C07299=1201.036,66.508,-47.398,-179.072,5.766,148.745
C07300=1201.040,66.258,-47.381,-179.075,5.765,148.746
C07301=1201.046,66.009,-47.364,-179.078,5.764,148.746
C07302=1201.050,65.759,-47.347,-179.080,5.763,148.747
C07303=1201.056,65.510,-47.330,-179.083,5.762,148.747
C07304=1201.060,65.261,-47.313,-179.086,5.762,148.748
C07305=1201.065,65.012,-47.296,-179.088,5.761,148.748
C07306=1201.070,64.763,-47.279,-179.090,5.760,148.749
C07307=1201.075,64.513,-47.263,-179.093,5.760,148.750
C07308=1201.080,64.263,-47.245,-179.096,5.758,148.750
C07309=1201.085,64.014,-47.229,-179.098,5.757,148.751
C07310=1201.090,63.765,-47.212,-179.101,5.757,148.751
C07311=1201.095,63.515,-47.195,-179.103,5.756,148.752
C07312=1201.099,63.266,-47.178,-179.106,5.755,148.753
C07313=1201.104,63.017,-47.162,-179.109,5.754,148.753
C07314=1201.110,62.767,-47.145,-179.111,5.753,148.754
C07315=1201.114,62.518,-47.128,-179.114,5.753,148.754
C07316=1201.119,62.268,-47.111,-179.116,5.752,148.755
C07317=1201.124,62.019,-47.095,-179.119,5.751,148.756
C07318=1201.129,61.770,-47.078,-179.121,5.751,148.756
C07319=1201.134,61.519,-47.062,-179.124,5.749,148.757
C07320=1201.140,61.270,-47.045,-179.127,5.749,148.757
C07321=1201.144,61.021,-47.028,-179.129,5.748,148.758
C07322=1201.149,60.771,-47.012,-179.132,5.747,148.758
C07323=1201.154,60.522,-46.995,-179.134,5.747,148.759
C07324=1201.159,60.273,-46.978,-179.137,5.746,148.760
C07325=1201.164,60.024,-46.962,-179.140,5.744,148.760
C07326=1201.168,59.775,-46.945,-179.142,5.744,148.761
C07327=1201.174,59.525,-46.928,-179.145,5.743,148.761
C07328=1201.179,59.276,-46.912,-179.147,5.742,148.762
C07329=1201.183,59.026,-46.896,-179.150,5.742,148.763
C07330=1201.188,58.776,-46.879,-179.152,5.741,148.763
C07331=1201.194,58.527,-46.862,-179.155,5.740,148.764
C07332=1201.198,58.278,-46.845,-179.158,5.739,148.764
C07333=1201.203,58.029,-46.829,-179.160,5.738,148.765
C07334=1201.208,57.779,-46.813,-179.163,5.738,148.766
C07335=1201.213,57.529,-46.796,-179.165,5.737,148.766
C07336=1201.218,57.280,-46.780,-179.168,5.736,148.767
C07337=1201.223,57.031,-46.763,-179.170,5.736,148.767
C07338=1201.228,56.782,-46.747,-179.173,5.734,148.768
C07339=1201.233,56.532,-46.731,-179.176,5.734,148.769
C07340=1201.238,56.282,-46.713,-179.178,5.733,148.769
C07341=1201.243,56.033,-46.697,-179.181,5.732,148.770
C07342=1201.248,55.784,-46.680,-179.183,5.732,148.770
C07343=1201.253,55.534,-46.665,-179.186,5.731,148.771
C07344=1201.258,55.266,-46.647,-179.189,5.729,148.772
C07345=1201.264,54.997,-46.629,-179.191,5.729,148.772
C07346=1201.269,54.729,-46.611,-179.194,5.728,148.773
C07347=1201.274,54.460,-46.594,-179.197,5.727,148.774
C07348=1201.279,54.211,-46.578,-179.200,5.726,148.774
C07349=1201.284,53.962,-46.561,-179.202,5.726,148.775
C07350=1201.288,53.712,-46.545,-179.204,5.725,148.775
C07351=1201.294,53.463,-46.528,-179.207,5.724,148.776
C07352=1201.299,53.213,-46.512,-179.210,5.724,148.777
C07353=1201.304,52.964,-46.496,-179.212,5.723,148.777
C07354=1201.309,52.714,-46.479,-179.215,5.722,148.778
C07355=1201.314,52.465,-46.464,-179.218,5.721,148.778
C07356=1201.318,52.215,-46.447,-179.220,5.721,148.779
C07357=1201.324,51.967,-46.431,-179.223,5.720,148.780
C07358=1201.328,51.716,-46.415,-179.225,5.719,148.780
C07359=1201.333,51.468,-46.398,-179.228,5.719,148.781
C07360=1201.338,51.218,-46.383,-179.230,5.718,148.781
C07361=1201.343,50.969,-46.366,-179.233,5.717,148.782
C07362=1201.348,50.719,-46.350,-179.235,5.717,148.783
C07363=1201.353,50.470,-46.334,-179.238,5.716,148.783
C07364=1201.358,50.220,-46.317,-179.241,5.714,148.784
C07365=1201.364,49.971,-46.301,-179.243,5.714,148.784
C07366=1201.368,49.721,-46.284,-179.246,5.713,148.785
C07367=1201.374,49.472,-46.269,-179.249,5.713,148.786
C07368=1201.378,49.222,-46.252,-179.251,5.712,148.786
C07369=1201.383,48.973,-46.237,-179.253,5.711,148.787
C07370=1201.388,48.723,-46.220,-179.256,5.711,148.788
C07371=1201.393,48.474,-46.204,-179.258,5.710,148.788
C07372=1201.398,48.225,-46.188,-179.261,5.709,148.789
C07373=1201.403,47.975,-46.172,-179.264,5.708,148.789
C07374=1201.408,47.725,-46.156,-179.267,5.708,148.790
C07375=1201.412,47.477,-46.140,-179.269,5.707,148.790
C07376=1201.418,47.227,-46.125,-179.271,5.706,148.791
C07377=1201.422,46.978,-46.108,-179.274,5.706,148.792
C07378=1201.428,46.728,-46.093,-179.277,5.705,148.792
C07379=1201.432,46.479,-46.076,-179.279,5.704,148.793
C07380=1201.437,46.229,-46.060,-179.281,5.704,148.794
C07381=1201.442,45.979,-46.044,-179.284,5.703,148.794
C07382=1201.447,45.731,-46.028,-179.286,5.702,148.795
C07383=1201.453,45.481,-46.012,-179.289,5.702,148.795
C07384=1201.458,45.231,-45.997,-179.292,5.700,148.796
C07385=1201.463,44.982,-45.980,-179.295,5.700,148.797
C07386=1201.467,44.732,-45.964,-179.297,5.699,148.797
C07387=1201.472,44.483,-45.948,-179.300,5.698,148.798
C07388=1201.478,44.234,-45.932,-179.302,5.698,148.798
C07389=1201.482,43.984,-45.917,-179.305,5.697,148.799
C07390=1201.487,43.735,-45.901,-179.307,5.696,148.800
C07391=1201.492,43.485,-45.885,-179.310,5.696,148.800
C07392=1201.497,43.236,-45.869,-179.312,5.695,148.801
C07393=1201.503,42.986,-45.854,-179.315,5.695,148.802
C07394=1201.507,42.737,-45.837,-179.317,5.694,148.802
C07395=1201.512,42.488,-45.821,-179.320,5.693,148.803
C07396=1201.518,42.238,-45.806,-179.322,5.693,148.803
C07397=1201.522,41.988,-45.790,-179.325,5.692,148.804
C07398=1201.527,41.740,-45.774,-179.328,5.691,148.804
C07399=1201.532,41.490,-45.758,-179.330,5.690,148.805
C07400=1201.537,41.240,-45.743,-179.333,5.690,148.806
C07401=1201.542,40.991,-45.727,-179.336,5.689,148.806
C07402=1201.547,40.741,-45.710,-179.338,5.688,148.807
C07403=1201.552,40.492,-45.695,-179.340,5.688,148.808
C07404=1201.557,40.243,-45.680,-179.343,5.687,148.808
C07405=1201.562,39.993,-45.664,-179.346,5.687,148.809
C07406=1201.567,39.743,-45.648,-179.348,5.686,148.809
C07407=1201.572,39.494,-45.633,-179.350,5.685,148.810
C07408=1201.577,39.245,-45.617,-179.353,5.685,148.811
C07409=1201.582,38.995,-45.601,-179.356,5.684,148.811
C07410=1201.587,38.746,-45.585,-179.358,5.683,148.812
C07411=1201.592,38.496,-45.570,-179.361,5.683,148.813
C07412=1201.597,38.247,-45.554,-179.363,5.682,148.813
C07413=1201.602,37.997,-45.539,-179.366,5.682,148.814
C07414=1201.607,37.748,-45.523,-179.368,5.681,148.814
C07415=1201.612,37.498,-45.507,-179.371,5.680,148.815
C07416=1201.617,37.249,-45.492,-179.374,5.679,148.816
C07417=1201.622,37.000,-45.476,-179.376,5.678,148.816
C07418=1201.627,36.750,-45.460,-179.379,5.678,148.817
C07419=1201.631,36.501,-45.445,-179.381,5.677,148.817
C07420=1201.637,36.251,-45.429,-179.384,5.676,148.818
C07421=1201.642,36.002,-45.414,-179.387,5.676,148.819
C07422=1201.647,35.752,-45.398,-179.389,5.675,148.820
C07423=1201.651,35.503,-45.383,-179.391,5.674,148.820
C07424=1201.657,35.253,-45.367,-179.394,5.674,148.821
C07425=1201.662,35.004,-45.352,-179.397,5.673,148.821
C07426=1201.667,34.755,-45.337,-179.399,5.673,148.822
C07427=1201.672,34.505,-45.321,-179.401,5.672,148.822
C07428=1201.677,34.255,-45.305,-179.404,5.671,148.823
C07429=1201.682,34.006,-45.290,-179.407,5.671,148.824
C07430=1201.687,33.757,-45.275,-179.409,5.670,148.824
C07431=1201.691,33.507,-45.259,-179.412,5.670,148.825
C07432=1201.697,33.258,-45.244,-179.414,5.669,148.826
C07433=1201.702,33.008,-45.228,-179.417,5.668,148.826
C07434=1201.707,32.759,-45.213,-179.419,5.668,148.827
C07435=1201.712,32.510,-45.197,-179.422,5.667,148.828
C07436=1201.717,32.259,-45.182,-179.424,5.667,148.828
C07437=1201.722,32.010,-45.167,-179.427,5.666,148.829
C07438=1201.727,31.760,-45.152,-179.430,5.665,148.829
C07439=1201.732,31.511,-45.137,-179.432,5.665,148.830
C07440=1201.737,31.262,-45.121,-179.434,5.664,148.831
C07441=1201.742,31.012,-45.105,-179.437,5.664,148.831
C07442=1201.747,30.763,-45.090,-179.440,5.663,148.832
C07443=1201.752,30.513,-45.075,-179.442,5.663,148.833
C07444=1201.757,30.264,-45.060,-179.445,5.662,148.833
C07445=1201.762,30.014,-45.045,-179.447,5.661,148.834
C07446=1201.766,29.764,-45.029,-179.450,5.661,148.834
C07447=1201.772,29.515,-45.014,-179.452,5.660,148.835
C07448=1201.777,29.246,-44.998,-179.455,5.660,148.836
C07449=1201.782,28.978,-44.981,-179.458,5.658,148.836
C07450=1201.788,28.709,-44.965,-179.461,5.658,148.837
C07451=1201.793,28.441,-44.948,-179.464,5.657,148.838
C07452=1201.798,28.191,-44.933,-179.466,5.657,148.838
C07453=1201.803,27.941,-44.918,-179.469,5.656,148.839
C07454=1201.809,27.692,-44.903,-179.471,5.655,148.840
C07455=1201.813,27.443,-44.888,-179.474,5.655,148.840
C07456=1201.818,27.193,-44.872,-179.476,5.654,148.841
C07457=1201.823,26.943,-44.858,-179.479,5.654,148.842
C07458=1201.829,26.694,-44.842,-179.481,5.653,148.842
C07459=1201.833,26.445,-44.827,-179.484,5.652,148.843
C07460=1201.839,26.195,-44.812,-179.486,5.652,148.843
C07461=1201.844,25.946,-44.797,-179.489,5.651,148.844
C07462=1201.849,25.696,-44.782,-179.492,5.651,148.845
C07463=1201.854,25.447,-44.767,-179.494,5.650,148.845
C07464=1201.859,25.197,-44.752,-179.496,5.649,148.846
C07465=1201.863,24.947,-44.736,-179.499,5.649,148.847
C07466=1201.868,24.698,-44.721,-179.502,5.648,148.847
C07467=1201.874,24.448,-44.706,-179.504,5.648,148.848
C07468=1201.878,24.199,-44.691,-179.507,5.647,148.848
C07469=1201.884,23.950,-44.676,-179.509,5.646,148.849
C07470=1201.889,23.700,-44.662,-179.512,5.646,148.850
C07471=1201.893,23.451,-44.647,-179.514,5.645,148.850
C07472=1201.899,23.201,-44.632,-179.517,5.645,148.851
C07473=1201.904,22.952,-44.617,-179.519,5.645,148.852
C07474=1201.908,22.703,-44.602,-179.521,5.644,148.852
C07475=1201.914,22.453,-44.587,-179.524,5.644,148.853
C07476=1201.919,22.203,-44.572,-179.527,5.643,148.854
C07477=1201.924,21.953,-44.557,-179.529,5.643,148.854
C07478=1201.929,21.704,-44.542,-179.531,5.642,148.855
C07479=1201.933,21.454,-44.527,-179.534,5.641,148.855
C07480=1201.939,21.205,-44.512,-179.537,5.641,148.856
C07481=1201.943,20.955,-44.497,-179.539,5.640,148.857
C07482=1201.948,20.706,-44.483,-179.542,5.640,148.857
C07483=1201.954,20.456,-44.467,-179.544,5.639,148.858
C07484=1201.959,20.207,-44.453,-179.547,5.638,148.859
C07485=1201.963,19.958,-44.438,-179.549,5.638,148.859
C07486=1201.969,19.708,-44.423,-179.552,5.637,148.860
C07487=1201.974,19.458,-44.408,-179.555,5.637,148.861
C07488=1201.979,19.209,-44.394,-179.557,5.636,148.861
C07489=1201.984,18.959,-44.378,-179.560,5.636,148.862
C07490=1201.989,18.710,-44.364,-179.562,5.635,148.862
C07491=1201.994,18.460,-44.349,-179.565,5.634,148.863
C07492=1201.999,18.211,-44.334,-179.568,5.634,148.864
C07493=1202.004,17.961,-44.320,-179.570,5.633,148.864
C07494=1202.009,17.712,-44.305,-179.572,5.633,148.865
C07495=1202.014,17.462,-44.290,-179.575,5.632,148.866
C07496=1202.019,17.213,-44.275,-179.577,5.632,148.866
C07497=1202.024,16.963,-44.260,-179.580,5.632,148.867
C07498=1202.029,16.713,-44.246,-179.582,5.631,148.868
C07499=1202.034,16.464,-44.231,-179.585,5.630,148.868
C07500=1202.039,16.215,-44.217,-179.587,5.630,148.869
C07501=1202.045,15.966,-44.202,-179.590,5.629,148.869
C07502=1202.050,15.716,-44.187,-179.592,5.629,148.870
C07503=1202.055,15.466,-44.173,-179.595,5.628,148.871
C07504=1202.059,15.217,-44.158,-179.597,5.628,148.871
C07505=1202.064,14.967,-44.144,-179.600,5.627,148.872
C07506=1202.070,14.717,-44.129,-179.603,5.627,148.873
C07507=1202.075,14.468,-44.114,-179.605,5.626,148.873
C07508=1202.080,14.219,-44.100,-179.608,5.626,148.874
C07509=1202.085,13.969,-44.085,-179.611,5.625,148.875
C07510=1202.089,13.720,-44.070,-179.613,5.624,148.875
C07511=1202.095,13.470,-44.056,-179.615,5.624,148.876
C07512=1202.100,13.220,-44.041,-179.617,5.624,148.877
C07513=1202.105,12.970,-44.027,-179.620,5.623,148.877
C07514=1202.109,12.721,-44.012,-179.623,5.623,148.878
C07515=1202.115,12.472,-43.998,-179.625,5.622,148.878
C07516=1202.120,12.223,-43.984,-179.627,5.622,148.879
C07517=1202.125,11.973,-43.969,-179.630,5.621,148.880
C07518=1202.130,11.723,-43.954,-179.633,5.621,148.880
C07519=1202.135,11.474,-43.940,-179.635,5.620,148.881
C07520=1202.140,11.224,-43.925,-179.638,5.620,148.882
C07521=1202.145,10.974,-43.911,-179.640,5.619,148.882
C07522=1202.150,10.725,-43.896,-179.643,5.618,148.883
C07523=1202.155,10.476,-43.882,-179.646,5.618,148.884
C07524=1202.160,10.227,-43.868,-179.648,5.618,148.884
C07525=1202.165,9.977,-43.854,-179.650,5.617,148.885
C07526=1202.170,9.727,-43.839,-179.652,5.617,148.885
C07527=1202.175,9.477,-43.825,-179.655,5.616,148.886
C07528=1202.181,9.228,-43.809,-179.658,5.616,148.887
C07529=1202.185,8.978,-43.795,-179.660,5.615,148.888
C07530=1202.190,8.729,-43.781,-179.663,5.615,148.888
C07531=1202.196,8.480,-43.767,-179.666,5.614,148.889
C07532=1202.201,8.230,-43.753,-179.668,5.613,148.889
C07533=1202.206,7.980,-43.738,-179.671,5.613,148.890
C07534=1202.211,7.730,-43.724,-179.673,5.613,148.891
C07535=1202.216,7.481,-43.710,-179.675,5.613,148.891
C07536=1202.220,7.232,-43.695,-179.678,5.612,148.892
C07537=1202.226,6.983,-43.681,-179.681,5.612,148.893
C07538=1202.231,6.733,-43.667,-179.683,5.611,148.893
C07539=1202.236,6.483,-43.652,-179.685,5.610,148.894
C07540=1202.241,6.233,-43.638,-179.688,5.610,148.895
C07541=1202.246,5.984,-43.624,-179.691,5.609,148.895
C07542=1202.251,5.735,-43.610,-179.693,5.609,148.896
C07543=1202.256,5.485,-43.596,-179.696,5.608,148.897
C07544=1202.261,5.235,-43.581,-179.698,5.608,148.897
C07545=1202.266,4.986,-43.567,-179.700,5.608,148.898
C07546=1202.271,4.736,-43.553,-179.703,5.607,148.898
C07547=1202.277,4.487,-43.539,-179.705,5.607,148.899
C07548=1202.282,4.237,-43.525,-179.708,5.606,148.900
C07549=1202.287,3.987,-43.510,-179.711,5.606,148.901
C07550=1202.292,3.738,-43.496,-179.713,5.605,148.901
C07551=1202.297,3.489,-43.482,-179.716,5.604,148.902
C07552=1202.303,3.219,-43.467,-179.718,5.604,148.902
C07553=1202.308,2.951,-43.452,-179.721,5.603,148.903
C07554=1202.313,2.681,-43.437,-179.724,5.603,148.904
C07555=1202.319,2.412,-43.422,-179.726,5.602,148.904
C07556=1202.324,2.162,-43.407,-179.729,5.602,148.905
C07557=1202.328,1.913,-43.394,-179.731,5.602,148.906
C07558=1202.333,1.664,-43.380,-179.734,5.602,148.907
C07559=1202.338,1.414,-43.365,-179.736,5.601,148.907
C07560=1202.344,1.165,-43.351,-179.739,5.601,148.908
C07561=1202.349,0.915,-43.337,-179.741,5.600,148.908
C07562=1202.354,0.665,-43.323,-179.744,5.599,148.909
C07563=1202.359,0.415,-43.309,-179.746,5.599,148.910
C07564=1202.365,0.166,-43.295,-179.749,5.598,148.910
C07565=1202.370,-0.084,-43.281,-179.751,5.599,148.911
C07566=1202.374,-0.333,-43.267,-179.754,5.598,148.912
C07567=1202.379,-0.582,-43.254,-179.756,5.598,148.912
C07568=1202.384,-0.832,-43.239,-179.759,5.597,148.913
C07569=1202.389,-1.081,-43.225,-179.761,5.596,148.914
C07570=1202.394,-1.332,-43.211,-179.764,5.596,148.914
C07571=1202.400,-1.581,-43.198,-179.767,5.595,148.915
C07572=1202.404,-1.830,-43.184,-179.769,5.596,148.916
C07573=1202.409,-2.080,-43.170,-179.771,5.595,148.916
C07574=1202.415,-2.329,-43.156,-179.773,5.594,148.917
C07575=1202.420,-2.579,-43.142,-179.776,5.594,148.918
C07576=1202.425,-2.829,-43.128,-179.779,5.593,148.918
C07577=1202.430,-3.078,-43.115,-179.781,5.593,148.919
C07578=1202.435,-3.327,-43.100,-179.784,5.592,148.920
C07579=1202.440,-3.578,-43.087,-179.786,5.593,148.920
C07580=1202.446,-3.827,-43.073,-179.788,5.592,148.921
C07581=1202.450,-4.076,-43.059,-179.791,5.591,148.921
C07582=1202.455,-4.326,-43.046,-179.794,5.591,148.922
C07583=1202.461,-4.575,-43.032,-179.796,5.590,148.923
C07584=1202.466,-4.825,-43.017,-179.799,5.590,148.924
C07585=1202.470,-5.075,-43.004,-179.801,5.590,148.924
C07586=1202.476,-5.324,-42.990,-179.804,5.590,148.925
C07587=1202.481,-5.574,-42.976,-179.806,5.589,148.925
C07588=1202.486,-5.823,-42.962,-179.808,5.588,148.926
C07589=1202.491,-6.073,-42.949,-179.811,5.588,148.927
C07590=1202.496,-6.323,-42.935,-179.814,5.587,148.927
C07591=1202.501,-6.572,-42.921,-179.816,5.588,148.928
C07592=1202.506,-6.822,-42.908,-179.819,5.587,148.929
C07593=1202.511,-7.071,-42.894,-179.821,5.586,148.929
C07594=1202.517,-7.321,-42.881,-179.823,5.586,148.930
C07595=1202.521,-7.571,-42.866,-179.826,5.585,148.931
C07596=1202.526,-7.819,-42.853,-179.829,5.585,148.931
C07597=1202.532,-8.070,-42.840,-179.831,5.585,148.932
C07598=1202.537,-8.319,-42.825,-179.833,5.585,148.933
C07599=1202.542,-8.569,-42.813,-179.836,5.584,148.933
C07600=1202.547,-8.818,-42.798,-179.838,5.583,148.934
C07601=1202.552,-9.067,-42.784,-179.841,5.583,148.935
C07602=1202.557,-9.317,-42.771,-179.844,5.582,148.935
C07603=1202.562,-9.566,-42.758,-179.846,5.583,148.936
C07604=1202.567,-9.817,-42.744,-179.848,5.582,148.937
C07605=1202.572,-10.066,-42.730,-179.851,5.582,148.937
C07606=1202.578,-10.316,-42.717,-179.854,5.581,148.938
C07607=1202.582,-10.565,-42.703,-179.856,5.580,148.938
C07608=1202.588,-10.815,-42.690,-179.858,5.580,148.939
C07609=1202.593,-11.065,-42.676,-179.860,5.580,148.940
C07610=1202.598,-11.314,-42.663,-179.863,5.580,148.941
C07611=1202.603,-11.564,-42.649,-179.866,5.579,148.941
C07612=1202.607,-11.814,-42.636,-179.868,5.579,148.942
C07613=1202.613,-12.063,-42.622,-179.871,5.578,148.942
C07614=1202.618,-12.313,-42.609,-179.873,5.578,148.943
C07615=1202.623,-12.562,-42.595,-179.875,5.578,148.944
C07616=1202.628,-12.812,-42.582,-179.878,5.577,148.944
C07617=1202.633,-13.061,-42.568,-179.881,5.577,148.945
C07618=1202.638,-13.311,-42.555,-179.883,5.576,148.946
C07619=1202.643,-13.560,-42.542,-179.885,5.576,148.947
C07620=1202.648,-13.810,-42.528,-179.888,5.576,148.947
C07621=1202.653,-14.059,-42.515,-179.890,5.575,148.948
C07622=1202.658,-14.309,-42.501,-179.893,5.575,148.948
C07623=1202.664,-14.559,-42.488,-179.896,5.574,148.949
C07624=1202.668,-14.808,-42.474,-179.898,5.574,148.950
C07625=1202.674,-15.058,-42.461,-179.900,5.574,148.951
C07626=1202.679,-15.308,-42.448,-179.903,5.574,148.951
C07627=1202.684,-15.557,-42.434,-179.905,5.573,148.952
C07628=1202.689,-15.807,-42.421,-179.908,5.572,148.952
C07629=1202.695,-16.056,-42.408,-179.910,5.572,148.953
C07630=1202.699,-16.306,-42.394,-179.912,5.572,148.954
C07631=1202.705,-16.555,-42.381,-179.915,5.572,148.954
C07632=1202.709,-16.805,-42.368,-179.918,5.571,148.955
C07633=1202.715,-17.054,-42.354,-179.920,5.571,148.956
C07634=1202.720,-17.304,-42.342,-179.922,5.571,148.956
C07635=1202.725,-17.554,-42.328,-179.925,5.570,148.957
C07636=1202.730,-17.803,-42.315,-179.927,5.570,148.958
C07637=1202.735,-18.053,-42.302,-179.930,5.569,148.958
C07638=1202.740,-18.302,-42.289,-179.933,5.569,148.959
C07639=1202.745,-18.552,-42.276,-179.935,5.569,148.960
C07640=1202.751,-18.801,-42.262,-179.937,5.568,148.960
C07641=1202.755,-19.051,-42.249,-179.940,5.568,148.961
C07642=1202.761,-19.301,-42.236,-179.942,5.567,148.962
C07643=1202.766,-19.550,-42.223,-179.944,5.567,148.962
C07644=1202.771,-19.800,-42.209,-179.947,5.567,148.963
C07645=1202.776,-20.049,-42.196,-179.950,5.566,148.964
C07646=1202.781,-20.299,-42.183,-179.952,5.566,148.964
C07647=1202.787,-20.549,-42.170,-179.955,5.566,148.965
C07648=1202.792,-20.798,-42.157,-179.957,5.565,148.966
C07649=1202.797,-21.048,-42.143,-179.959,5.565,148.966
C07650=1202.802,-21.297,-42.130,-179.962,5.565,148.967
C07651=1202.806,-21.547,-42.118,-179.964,5.564,148.968
C07652=1202.812,-21.797,-42.104,-179.967,5.564,148.968
C07653=1202.817,-22.046,-42.092,-179.969,5.564,148.969
C07654=1202.821,-22.296,-42.078,-179.972,5.563,148.970
C07655=1202.827,-22.545,-42.065,-179.974,5.563,148.970
C07656=1202.832,-22.815,-42.051,-179.977,5.562,148.971
C07657=1202.838,-23.085,-42.037,-179.980,5.562,148.972
C07658=1202.844,-23.355,-42.023,-179.982,5.562,148.973
C07659=1202.849,-23.624,-42.009,-179.985,5.562,148.973
C07660=1202.854,-23.873,-41.996,-179.987,5.561,148.974
C07661=1202.859,-24.123,-41.982,-179.989,5.561,148.974
C07662=1202.865,-24.373,-41.970,-179.992,5.560,148.975
C07663=1202.870,-24.622,-41.957,-179.994,5.560,148.976
C07664=1202.875,-24.872,-41.944,-179.997,5.560,148.976
C07665=1202.880,-25.122,-41.931,-180.000,5.559,148.977
C07666=1202.885,-25.371,-41.918,179.998,5.559,148.978
C07667=1202.890,-25.621,-41.905,179.996,5.559,148.979
C07668=1202.896,-25.871,-41.892,179.994,5.558,148.979
C07669=1202.900,-26.121,-41.879,179.991,5.558,148.980
C07670=1202.905,-26.370,-41.867,179.988,5.558,148.980
C07671=1202.911,-26.620,-41.854,179.986,5.558,148.981
C07672=1202.916,-26.869,-41.841,179.984,5.557,148.982
C07673=1202.921,-27.119,-41.828,179.981,5.557,148.983
C07674=1202.926,-27.368,-41.815,179.978,5.556,148.983
C07675=1202.932,-27.618,-41.802,179.976,5.557,148.984
C07676=1202.936,-27.868,-41.789,179.974,5.556,148.984
C07677=1202.941,-28.117,-41.777,179.971,5.555,148.985
C07678=1202.947,-28.366,-41.764,179.969,5.555,148.986
C07679=1202.951,-28.616,-41.751,179.967,5.555,148.986
C07680=1202.957,-28.866,-41.738,179.964,5.555,148.987
C07681=1202.962,-29.115,-41.725,179.961,5.554,148.988
C07682=1202.967,-29.365,-41.712,179.959,5.554,148.989
C07683=1202.972,-29.615,-41.700,179.957,5.554,148.989
C07684=1202.978,-29.864,-41.686,179.954,5.553,148.990
C07685=1202.983,-30.114,-41.674,179.952,5.553,148.990
C07686=1202.987,-30.364,-41.661,179.949,5.552,148.991
C07687=1202.992,-30.613,-41.648,179.947,5.553,148.992
C07688=1202.997,-30.862,-41.636,179.944,5.552,148.993
C07689=1203.003,-31.112,-41.623,179.942,5.552,148.993
C07690=1203.008,-31.363,-41.610,179.939,5.551,148.994
C07691=1203.013,-31.612,-41.598,179.937,5.551,148.994
C07692=1203.018,-31.861,-41.585,179.935,5.551,148.995
C07693=1203.024,-32.111,-41.572,179.932,5.550,148.996
C07694=1203.028,-32.361,-41.559,179.929,5.550,148.996
C07695=1203.033,-32.610,-41.547,179.927,5.550,148.997
C07696=1203.038,-32.859,-41.534,179.925,5.550,148.998
C07697=1203.044,-33.109,-41.522,179.922,5.549,148.998
C07698=1203.049,-33.360,-41.509,179.920,5.549,148.999
C07699=1203.054,-33.609,-41.496,179.918,5.549,149.000
C07700=1203.059,-33.858,-41.484,179.915,5.548,149.000
C07701=1203.064,-34.107,-41.471,179.912,5.548,149.001
C07702=1203.070,-34.357,-41.459,179.910,5.548,149.002
C07703=1203.074,-34.607,-41.446,179.908,5.548,149.003
C07704=1203.079,-34.857,-41.434,179.905,5.547,149.003
C07705=1203.085,-35.106,-41.421,179.903,5.547,149.004
C07706=1203.091,-35.356,-41.409,179.901,5.547,149.004
C07707=1203.096,-35.606,-41.396,179.898,5.546,149.005
C07708=1203.100,-35.856,-41.383,179.895,5.546,149.006
C07709=1203.105,-36.105,-41.370,179.893,5.546,149.006
C07710=1203.111,-36.355,-41.358,179.891,5.546,149.007
C07711=1203.116,-36.604,-41.346,179.888,5.545,149.008
C07712=1203.121,-36.854,-41.333,179.886,5.545,149.008
C07713=1203.126,-37.104,-41.320,179.884,5.545,149.009
C07714=1203.131,-37.353,-41.308,179.881,5.544,149.010
C07715=1203.136,-37.603,-41.296,179.878,5.544,149.010
C07716=1203.141,-37.852,-41.283,179.876,5.544,149.011
C07717=1203.147,-38.102,-41.271,179.874,5.544,149.012
C07718=1203.152,-38.351,-41.259,179.871,5.543,149.012
C07719=1203.157,-38.601,-41.246,179.869,5.543,149.013
C07720=1203.162,-38.851,-41.234,179.867,5.543,149.014
C07721=1203.167,-39.101,-41.221,179.864,5.542,149.014
C07722=1203.172,-39.350,-41.209,179.861,5.542,149.015
C07723=1203.178,-39.600,-41.197,179.859,5.542,149.016
C07724=1203.183,-39.849,-41.184,179.857,5.542,149.017
C07725=1203.188,-40.099,-41.172,179.855,5.541,149.017
C07726=1203.193,-40.348,-41.160,179.852,5.541,149.018
C07727=1203.198,-40.598,-41.147,179.850,5.541,149.018
C07728=1203.203,-40.848,-41.135,179.847,5.540,149.019
C07729=1203.208,-41.098,-41.122,179.845,5.541,149.020
C07730=1203.214,-41.348,-41.110,179.842,5.540,149.021
C07731=1203.219,-41.597,-41.098,179.840,5.540,149.021
C07732=1203.224,-41.846,-41.085,179.838,5.539,149.022
C07733=1203.229,-42.096,-41.073,179.835,5.539,149.022
C07734=1203.235,-42.346,-41.061,179.833,5.539,149.023
C07735=1203.240,-42.595,-41.049,179.830,5.538,149.024
C07736=1203.244,-42.846,-41.036,179.828,5.539,149.024
C07737=1203.249,-43.095,-41.025,179.825,5.538,149.025
C07738=1203.254,-43.344,-41.012,179.823,5.538,149.026
C07739=1203.260,-43.594,-41.000,179.821,5.538,149.026
C07740=1203.265,-43.844,-40.987,179.818,5.537,149.027
C07741=1203.270,-44.094,-40.976,179.816,5.537,149.028
C07742=1203.275,-44.343,-40.963,179.814,5.537,149.028
C07743=1203.281,-44.593,-40.951,179.811,5.537,149.029
C07744=1203.286,-44.842,-40.938,179.808,5.536,149.030
C07745=1203.291,-45.092,-40.927,179.806,5.535,149.030
C07746=1203.296,-45.341,-40.915,179.804,5.536,149.031
C07747=1203.301,-45.591,-40.903,179.801,5.535,149.032
C07748=1203.306,-45.840,-40.890,179.799,5.535,149.032
C07749=1203.312,-46.090,-40.878,179.797,5.535,149.033
C07750=1203.317,-46.340,-40.866,179.794,5.535,149.034
C07751=1203.322,-46.590,-40.854,179.791,5.534,149.035
C07752=1203.327,-46.840,-40.841,179.790,5.534,149.035
C07753=1203.332,-47.089,-40.829,179.787,5.534,149.036
C07754=1203.337,-47.339,-40.818,179.784,5.533,149.036
C07755=1203.342,-47.589,-40.806,179.782,5.534,149.037
C07756=1203.347,-47.838,-40.793,179.780,5.533,149.038
C07757=1203.353,-48.088,-40.781,179.777,5.533,149.039
C07758=1203.357,-48.337,-40.769,179.775,5.533,149.039
C07759=1203.363,-48.587,-40.757,179.773,5.532,149.040
C07760=1203.369,-48.857,-40.745,179.770,5.532,149.040
C07761=1203.375,-49.128,-40.731,179.767,5.532,149.041
C07762=1203.380,-49.398,-40.718,179.765,5.532,149.042
C07763=1203.386,-49.668,-40.706,179.762,5.532,149.043
C07764=1203.391,-49.917,-40.693,179.760,5.531,149.043
C07765=1203.396,-50.167,-40.682,179.757,5.530,149.044
C07766=1203.401,-50.417,-40.670,179.755,5.531,149.045
C07767=1203.406,-50.666,-40.657,179.753,5.530,149.045
C07768=1203.412,-50.916,-40.645,179.750,5.530,149.046
C07769=1203.416,-51.165,-40.634,179.748,5.530,149.047
C07770=1203.422,-51.415,-40.621,179.745,5.530,149.047
C07771=1203.427,-51.665,-40.610,179.743,5.529,149.048
C07772=1203.432,-51.915,-40.598,179.741,5.529,149.049
C07773=1203.437,-52.164,-40.586,179.738,5.529,149.049
C07774=1203.442,-52.414,-40.574,179.736,5.529,149.050
C07775=1203.448,-52.663,-40.562,179.734,5.529,149.051
C07776=1203.452,-52.913,-40.551,179.731,5.528,149.051
C07777=1203.458,-53.163,-40.539,179.729,5.529,149.052
C07778=1203.463,-53.412,-40.526,179.727,5.528,149.053
C07779=1203.468,-53.662,-40.515,179.724,5.527,149.053
C07780=1203.473,-53.912,-40.503,179.722,5.528,149.054
C07781=1203.478,-54.162,-40.491,179.719,5.527,149.055
C07782=1203.483,-54.411,-40.480,179.717,5.527,149.055
C07783=1203.489,-54.660,-40.468,179.714,5.527,149.056
C07784=1203.494,-54.910,-40.456,179.712,5.526,149.057
C07785=1203.499,-55.160,-40.444,179.710,5.526,149.057
C07786=1203.504,-55.410,-40.432,179.708,5.526,149.058
C07787=1203.510,-55.660,-40.421,179.705,5.526,149.059
C07788=1203.515,-55.909,-40.409,179.702,5.525,149.059
C07789=1203.520,-56.158,-40.397,179.700,5.526,149.060
C07790=1203.525,-56.408,-40.385,179.697,5.525,149.061
C07791=1203.530,-56.658,-40.374,179.695,5.524,149.061
C07792=1203.535,-56.908,-40.362,179.693,5.525,149.062
C07793=1203.540,-57.158,-40.350,179.690,5.524,149.063
C07794=1203.545,-57.408,-40.338,179.688,5.525,149.063
C07795=1203.551,-57.657,-40.327,179.686,5.524,149.064
C07796=1203.556,-57.906,-40.316,179.683,5.524,149.065
C07797=1203.561,-58.156,-40.304,179.681,5.524,149.065
C07798=1203.566,-58.405,-40.292,179.679,5.523,149.066
C07799=1203.571,-58.655,-40.280,179.676,5.523,149.067
C07800=1203.577,-58.905,-40.268,179.674,5.523,149.067
C07801=1203.581,-59.155,-40.257,179.671,5.523,149.068
C07802=1203.587,-59.405,-40.245,179.669,5.522,149.069
C07803=1203.592,-59.654,-40.234,179.667,5.522,149.069
C07804=1203.598,-59.904,-40.222,179.664,5.522,149.070
C07805=1203.602,-60.153,-40.211,179.662,5.522,149.071
C07806=1203.608,-60.403,-40.199,179.660,5.522,149.071
C07807=1203.613,-60.653,-40.187,179.657,5.521,149.072
C07808=1203.618,-60.903,-40.176,179.655,5.522,149.073
C07809=1203.624,-61.152,-40.164,179.653,5.521,149.073
C07810=1203.629,-61.402,-40.153,179.650,5.520,149.074
C07811=1203.634,-61.652,-40.141,179.648,5.521,149.075
C07812=1203.639,-61.901,-40.130,179.645,5.520,149.075
C07813=1203.644,-62.151,-40.118,179.643,5.521,149.076
C07814=1203.649,-62.401,-40.106,179.641,5.520,149.077
C07815=1203.655,-62.650,-40.095,179.638,5.519,149.077
C07816=1203.659,-62.900,-40.084,179.636,5.520,149.078
C07817=1203.665,-63.150,-40.072,179.634,5.519,149.079
C07818=1203.670,-63.399,-40.060,179.631,5.519,149.079
C07819=1203.675,-63.649,-40.049,179.629,5.519,149.080
C07820=1203.681,-63.899,-40.038,179.626,5.519,149.081
C07821=1203.686,-64.149,-40.027,179.625,5.519,149.081
C07822=1203.691,-64.398,-40.015,179.622,5.518,149.082
C07823=1203.696,-64.648,-40.003,179.619,5.518,149.083
C07824=1203.701,-64.898,-39.992,179.617,5.518,149.083
C07825=1203.706,-65.147,-39.981,179.615,5.518,149.084
C07826=1203.712,-65.397,-39.969,179.612,5.517,149.085
C07827=1203.716,-65.646,-39.958,179.610,5.517,149.085
C07828=1203.722,-65.896,-39.946,179.608,5.517,149.086
C07829=1203.727,-66.146,-39.935,179.606,5.517,149.087
C07830=1203.733,-66.396,-39.924,179.603,5.517,149.087
C07831=1203.737,-66.645,-39.913,179.600,5.516,149.088
C07832=1203.743,-66.895,-39.901,179.598,5.517,149.089
C07833=1203.748,-67.145,-39.890,179.596,5.516,149.089
C07834=1203.753,-67.394,-39.879,179.594,5.516,149.090
C07835=1203.759,-67.644,-39.867,179.591,5.516,149.091
C07836=1203.763,-67.894,-39.856,179.589,5.515,149.091
C07837=1203.769,-68.144,-39.844,179.586,5.516,149.092
C07838=1203.774,-68.393,-39.833,179.584,5.515,149.093
C07839=1203.779,-68.642,-39.822,179.582,5.515,149.093
C07840=1203.784,-68.893,-39.811,179.580,5.515,149.094
C07841=1203.790,-69.142,-39.800,179.577,5.514,149.095
C07842=1203.794,-69.392,-39.789,179.575,5.515,149.095
C07843=1203.800,-69.641,-39.777,179.572,5.514,149.096
C07844=1203.805,-69.892,-39.766,179.570,5.514,149.097
C07845=1203.811,-70.141,-39.755,179.568,5.514,149.097
C07846=1203.816,-70.391,-39.743,179.565,5.513,149.098
C07847=1203.820,-70.640,-39.732,179.563,5.514,149.099
C07848=1203.827,-70.890,-39.721,179.560,5.513,149.099
C07849=1203.831,-71.140,-39.710,179.558,5.514,149.100
C07850=1203.836,-71.389,-39.699,179.556,5.513,149.101
C07851=1203.842,-71.640,-39.688,179.553,5.512,149.101
C07852=1203.847,-71.889,-39.677,179.551,5.513,149.102
C07853=1203.852,-72.138,-39.665,179.549,5.512,149.103
C07854=1203.857,-72.389,-39.654,179.547,5.513,149.104
C07855=1203.863,-72.638,-39.643,179.544,5.512,149.104
C07856=1203.867,-72.888,-39.632,179.542,5.511,149.105
C07857=1203.872,-73.138,-39.621,179.540,5.512,149.105
C07858=1203.878,-73.387,-39.610,179.537,5.511,149.106
C07859=1203.883,-73.637,-39.599,179.535,5.512,149.107
C07860=1203.888,-73.887,-39.588,179.533,5.511,149.107
C07861=1203.894,-74.136,-39.576,179.530,5.511,149.108
C07862=1203.899,-74.386,-39.565,179.528,5.511,149.109
C07863=1203.904,-74.635,-39.555,179.525,5.510,149.109
C07864=1203.910,-74.906,-39.543,179.523,5.511,149.110
C07865=1203.916,-75.177,-39.530,179.521,5.510,149.111
C07866=1203.921,-75.447,-39.519,179.518,5.510,149.112
C07867=1203.927,-75.718,-39.507,179.515,5.510,149.112
C07868=1203.931,-75.968,-39.496,179.513,5.510,149.113
C07869=1203.938,-76.218,-39.485,179.510,5.509,149.114
C07870=1203.942,-76.467,-39.474,179.508,5.510,149.114
C07871=1203.947,-76.718,-39.463,179.506,5.509,149.115
C07872=1203.953,-76.966,-39.452,179.504,5.509,149.116
C07873=1203.959,-77.217,-39.441,179.501,5.509,149.116
C07874=1203.964,-77.466,-39.430,179.499,5.509,149.117
C07875=1203.969,-77.716,-39.419,179.497,5.509,149.118
C07876=1203.974,-77.966,-39.408,179.494,5.508,149.118
C07877=1203.979,-78.215,-39.397,179.492,5.508,149.119
C07878=1203.985,-78.465,-39.386,179.490,5.508,149.120
C07879=1203.990,-78.714,-39.375,179.488,5.508,149.120
C07880=1203.995,-78.964,-39.364,179.485,5.508,149.121
C07881=1204.000,-79.214,-39.353,179.483,5.507,149.121
C07882=1204.005,-79.464,-39.343,179.481,5.507,149.122
C07883=1204.010,-79.714,-39.332,179.478,5.507,149.123
C07884=1204.016,-79.963,-39.321,179.476,5.507,149.124
C07885=1204.021,-80.213,-39.310,179.473,5.507,149.124
C07886=1204.026,-80.462,-39.299,179.472,5.507,149.125
C07887=1204.031,-80.713,-39.289,179.469,5.507,149.126
C07888=1204.036,-80.962,-39.278,179.466,5.506,149.126
C07889=1204.042,-81.212,-39.267,179.464,5.507,149.127
C07890=1204.046,-81.461,-39.256,179.462,5.506,149.128
C07891=1204.053,-81.711,-39.245,179.460,5.506,149.128
C07892=1204.058,-81.961,-39.235,179.457,5.506,149.129
C07893=1204.063,-82.210,-39.224,179.455,5.506,149.130
C07894=1204.068,-82.461,-39.213,179.453,5.506,149.130
C07895=1204.073,-82.710,-39.202,179.450,5.505,149.131
C07896=1204.078,-82.960,-39.192,179.448,5.505,149.131
C07897=1204.083,-83.210,-39.181,179.446,5.505,149.132
C07898=1204.089,-83.459,-39.170,179.444,5.505,149.133
C07899=1204.094,-83.709,-39.160,179.441,5.505,149.134
C07900=1204.099,-83.959,-39.149,179.439,5.505,149.134
C07901=1204.104,-84.208,-39.138,179.437,5.504,149.135
C07902=1204.109,-84.458,-39.128,179.434,5.505,149.135
C07903=1204.114,-84.708,-39.117,179.432,5.504,149.136
C07904=1204.121,-84.957,-39.106,179.429,5.504,149.137
C07905=1204.126,-85.208,-39.095,179.428,5.504,149.137
C07906=1204.131,-85.457,-39.085,179.425,5.503,149.138
C07907=1204.136,-85.707,-39.074,179.423,5.504,149.139
C07908=1204.141,-85.956,-39.063,179.420,5.503,149.140
C07909=1204.146,-86.207,-39.053,179.419,5.503,149.140
C07910=1204.152,-86.455,-39.042,179.416,5.503,149.141
C07911=1204.157,-86.706,-39.031,179.414,5.503,149.141
C07912=1204.162,-86.955,-39.021,179.411,5.503,149.142
C07913=1204.167,-87.206,-39.011,179.408,5.502,149.143
C07914=1204.173,-87.454,-39.000,179.407,5.502,149.143
C07915=1204.178,-87.705,-38.989,179.404,5.502,149.144
C07916=1204.183,-87.954,-38.979,179.402,5.502,149.145
C07917=1204.188,-88.204,-38.968,179.399,5.502,149.145
C07918=1204.193,-88.453,-38.957,179.397,5.502,149.146
C07919=1204.198,-88.704,-38.947,179.395,5.501,149.147
C07920=1204.204,-88.953,-38.937,179.393,5.502,149.147
C07921=1204.209,-89.203,-38.926,179.390,5.501,149.148
C07922=1204.214,-89.452,-38.915,179.388,5.501,149.149
C07923=1204.220,-89.702,-38.905,179.386,5.501,149.149
C07924=1204.225,-89.952,-38.894,179.383,5.501,149.150
C07925=1204.230,-90.201,-38.885,179.381,5.501,149.151
C07926=1204.235,-90.452,-38.874,179.379,5.500,149.151
C07927=1204.240,-90.701,-38.864,179.377,5.500,149.152
C07928=1204.245,-90.951,-38.853,179.374,5.500,149.153
C07929=1204.251,-91.200,-38.842,179.372,5.500,149.153
C07930=1204.256,-91.450,-38.832,179.370,5.500,149.154
C07931=1204.261,-91.700,-38.822,179.368,5.500,149.155
C07932=1204.267,-91.950,-38.811,179.365,5.500,149.155
C07933=1204.272,-92.200,-38.801,179.363,5.500,149.156
C07934=1204.277,-92.449,-38.791,179.361,5.500,149.157
C07935=1204.282,-92.699,-38.779,179.358,5.499,149.157
C07936=1204.288,-92.949,-38.769,179.356,5.499,149.158
C07937=1204.293,-93.198,-38.760,179.354,5.499,149.159
C07938=1204.298,-93.448,-38.749,179.352,5.499,149.159
C07939=1204.303,-93.698,-38.739,179.349,5.499,149.160
C07940=1204.308,-93.948,-38.728,179.347,5.499,149.160
C07941=1204.314,-94.197,-38.718,179.345,5.498,149.161
C07942=1204.319,-94.447,-38.708,179.343,5.499,149.162
C07943=1204.324,-94.697,-38.697,179.340,5.498,149.163
C07944=1204.330,-94.947,-38.687,179.338,5.498,149.163
C07945=1204.335,-95.196,-38.677,179.336,5.498,149.164
C07946=1204.340,-95.446,-38.667,179.333,5.498,149.164
C07947=1204.345,-95.696,-38.657,179.331,5.498,149.165
C07948=1204.350,-95.946,-38.646,179.329,5.498,149.166
C07949=1204.356,-96.195,-38.635,179.327,5.497,149.166
C07950=1204.361,-96.445,-38.625,179.324,5.498,149.167
C07951=1204.366,-96.694,-38.615,179.322,5.497,149.168
C07952=1204.371,-96.944,-38.605,179.320,5.496,149.168
C07953=1204.377,-97.194,-38.595,179.317,5.497,149.169
C07954=1204.382,-97.444,-38.585,179.315,5.496,149.170
C07955=1204.388,-97.694,-38.574,179.313,5.497,149.170
C07956=1204.393,-97.943,-38.564,179.311,5.496,149.171
C07957=1204.398,-98.193,-38.554,179.308,5.496,149.172
C07958=1204.403,-98.443,-38.544,179.306,5.496,149.172
C07959=1204.409,-98.692,-38.534,179.304,5.496,149.173
C07960=1204.414,-98.943,-38.523,179.301,5.496,149.174
C07961=1204.419,-99.192,-38.513,179.299,5.496,149.174
C07962=1204.424,-99.442,-38.503,179.297,5.496,149.175
C07963=1204.429,-99.692,-38.493,179.295,5.496,149.176
C07964=1204.435,-99.941,-38.483,179.292,5.495,149.176
C07965=1204.440,-100.191,-38.472,179.290,5.495,149.177
C07966=1204.445,-100.441,-38.462,179.288,5.495,149.178
C07967=1204.450,-100.690,-38.452,179.286,5.495,149.178
C07968=1204.455,-100.962,-38.441,179.283,5.495,149.179
C07969=1204.462,-101.233,-38.431,179.280,5.495,149.180
C07970=1204.468,-101.504,-38.420,179.278,5.495,149.180
C07971=1204.473,-101.776,-38.408,179.275,5.495,149.181
C07972=1204.478,-102.025,-38.399,179.274,5.495,149.182
C07973=1204.484,-102.275,-38.389,179.271,5.494,149.182
C07974=1204.489,-102.525,-38.378,179.269,5.495,149.183
C07975=1204.494,-102.775,-38.369,179.267,5.494,149.184
C07976=1204.500,-103.024,-38.359,179.265,5.494,149.184
C07977=1204.505,-103.275,-38.348,179.262,5.494,149.185
C07978=1204.510,-103.524,-38.339,179.260,5.494,149.186
C07979=1204.515,-103.773,-38.329,179.258,5.493,149.186
C07980=1204.521,-104.024,-38.319,179.256,5.494,149.187
C07981=1204.526,-104.274,-38.308,179.253,5.493,149.188
C07982=1204.531,-104.523,-38.299,179.251,5.494,149.188
C07983=1204.536,-104.773,-38.289,179.249,5.493,149.189
C07984=1204.542,-105.022,-38.278,179.246,5.492,149.190
C07985=1204.547,-105.273,-38.269,179.244,5.493,149.190
C07986=1204.552,-105.522,-38.259,179.242,5.492,149.191
C07987=1204.557,-105.772,-38.249,179.240,5.492,149.191
C07988=1204.563,-106.021,-38.239,179.237,5.492,149.192
C07989=1204.568,-106.272,-38.229,179.235,5.492,149.193
C07990=1204.573,-106.521,-38.220,179.233,5.492,149.193
C07991=1204.578,-106.771,-38.209,179.231,5.492,149.194
C07992=1204.584,-107.020,-38.199,179.228,5.492,149.195
C07993=1204.589,-107.270,-38.190,179.226,5.492,149.195
C07994=1204.594,-107.520,-38.180,179.224,5.491,149.196
C07995=1204.599,-107.770,-38.170,179.222,5.492,149.197
C07996=1204.605,-108.019,-38.160,179.219,5.491,149.197
C07997=1204.611,-108.269,-38.150,179.217,5.491,149.198
C07998=1204.615,-108.519,-38.141,179.215,5.491,149.199
C07999=1204.620,-108.769,-38.130,179.213,5.491,149.199
C08000=1204.626,-109.019,-38.121,179.210,5.490,149.200
C08001=1204.631,-109.268,-38.111,179.208,5.491,149.200
C08002=1204.637,-109.518,-38.101,179.206,5.491,149.201
C08003=1204.642,-109.768,-38.092,179.204,5.491,149.202
C08004=1204.647,-110.018,-38.081,179.202,5.491,149.202
C08005=1204.652,-110.267,-38.072,179.199,5.490,149.203
C08006=1204.658,-110.517,-38.062,179.197,5.491,149.204
C08007=1204.663,-110.766,-38.053,179.195,5.490,149.204
C08008=1204.668,-111.017,-38.043,179.193,5.490,149.205
C08009=1204.673,-111.266,-38.034,179.190,5.490,149.206
C08010=1204.678,-111.516,-38.023,179.189,5.490,149.206
C08011=1204.684,-111.766,-38.014,179.186,5.490,149.207
C08012=1204.689,-112.015,-38.004,179.184,5.490,149.208
C08013=1204.695,-112.266,-37.994,179.181,5.490,149.208
C08014=1204.700,-112.515,-37.985,179.180,5.490,149.209
C08015=1204.705,-112.764,-37.975,179.177,5.489,149.210
C08016=1204.710,-113.015,-37.965,179.175,5.489,149.210
C08017=1204.716,-113.265,-37.955,179.173,5.489,149.211
C08018=1204.721,-113.514,-37.946,179.171,5.489,149.211
C08019=1204.726,-113.764,-37.936,179.168,5.489,149.212
C08020=1204.732,-114.014,-37.927,179.166,5.489,149.213
C08021=1204.737,-114.263,-37.917,179.164,5.488,149.213
C08022=1204.742,-114.513,-37.908,179.162,5.489,149.214
C08023=1204.748,-114.763,-37.898,179.159,5.488,149.215
C08024=1204.752,-115.013,-37.888,179.157,5.488,149.215
C08025=1204.758,-115.263,-37.878,179.155,5.488,149.216
C08026=1204.763,-115.512,-37.869,179.153,5.488,149.217
C08027=1204.768,-115.762,-37.860,179.150,5.487,149.217
C08028=1204.774,-116.011,-37.850,179.148,5.488,149.218
C08029=1204.779,-116.261,-37.841,179.146,5.487,149.219
C08030=1204.785,-116.511,-37.831,179.144,5.487,149.219
C08031=1204.790,-116.761,-37.822,179.141,5.487,149.220
C08032=1204.796,-117.011,-37.812,179.139,5.487,149.221
C08033=1204.800,-117.260,-37.803,179.137,5.487,149.221
C08034=1204.806,-117.511,-37.793,179.135,5.487,149.222
C08035=1204.811,-117.760,-37.783,179.132,5.487,149.223
C08036=1204.816,-118.010,-37.774,179.131,5.487,149.223
C08037=1204.821,-118.260,-37.764,179.129,5.487,149.224
C08038=1204.827,-118.509,-37.755,179.126,5.487,149.224
C08039=1204.832,-118.760,-37.746,179.124,5.487,149.225
C08040=1204.837,-119.009,-37.736,179.122,5.486,149.226
C08041=1204.842,-119.259,-37.727,179.120,5.487,149.226
C08042=1204.848,-119.508,-37.717,179.117,5.486,149.227
C08043=1204.853,-119.758,-37.708,179.115,5.486,149.228
C08044=1204.858,-120.007,-37.698,179.113,5.486,149.228
C08045=1204.864,-120.257,-37.689,179.111,5.486,149.229
C08046=1204.869,-120.507,-37.680,179.108,5.485,149.229
C08047=1204.875,-120.757,-37.670,179.106,5.486,149.230
C08048=1204.880,-121.007,-37.661,179.104,5.485,149.231
C08049=1204.885,-121.257,-37.652,179.102,5.485,149.231
C08050=1204.890,-121.507,-37.641,179.099,5.485,149.232
C08051=1204.895,-121.757,-37.632,179.098,5.485,149.233
C08052=1204.900,-122.006,-37.624,179.095,5.485,149.233
C08053=1204.906,-122.256,-37.613,179.093,5.485,149.234
C08054=1204.911,-122.506,-37.604,179.091,5.485,149.234
C08055=1204.916,-122.756,-37.596,179.089,5.485,149.235
C08056=1204.922,-123.005,-37.585,179.087,5.485,149.236
C08057=1204.927,-123.255,-37.576,179.084,5.484,149.236
C08058=1204.932,-123.505,-37.568,179.082,5.485,149.237
C08059=1204.937,-123.754,-37.558,179.080,5.484,149.238
C08060=1204.943,-124.004,-37.548,179.078,5.484,149.238
C08061=1204.948,-124.254,-37.540,179.075,5.484,149.239
C08062=1204.953,-124.504,-37.531,179.074,5.484,149.240
C08063=1204.959,-124.754,-37.520,179.071,5.484,149.240
C08064=1204.964,-125.003,-37.512,179.069,5.484,149.241
C08065=1204.969,-125.253,-37.503,179.067,5.483,149.241
C08066=1204.974,-125.503,-37.494,179.065,5.484,149.242
C08067=1204.980,-125.753,-37.484,179.063,5.484,149.243
C08068=1204.985,-126.003,-37.475,179.060,5.483,149.243
C08069=1204.990,-126.252,-37.466,179.058,5.484,149.244
C08070=1204.996,-126.502,-37.457,179.056,5.483,149.245
C08071=1205.001,-126.752,-37.447,179.054,5.483,149.245
C08072=1204.580,-126.763,-37.485,179.050,5.486,149.247
C08073=1204.575,-126.513,-37.494,179.052,5.486,149.247
C08074=1204.570,-126.263,-37.503,179.054,5.487,149.246
C08075=1204.564,-126.013,-37.513,179.056,5.487,149.245
C08076=1204.559,-125.764,-37.522,179.059,5.487,149.245
C08077=1204.554,-125.514,-37.531,179.061,5.487,149.244
C08078=1204.548,-125.264,-37.541,179.062,5.487,149.244
C08079=1204.543,-125.014,-37.550,179.065,5.487,149.243
C08080=1204.538,-124.765,-37.559,179.067,5.487,149.242
C08081=1204.533,-124.515,-37.568,179.069,5.488,149.242
C08082=1204.527,-124.265,-37.578,179.071,5.487,149.241
C08083=1204.521,-124.015,-37.586,179.074,5.488,149.240
C08084=1204.517,-123.765,-37.596,179.076,5.487,149.240
C08085=1204.511,-123.515,-37.606,179.078,5.488,149.239
C08086=1204.506,-123.265,-37.614,179.080,5.487,149.238
C08087=1204.501,-123.016,-37.624,179.083,5.488,149.238
C08088=1204.495,-122.766,-37.633,179.085,5.488,149.237
C08089=1204.490,-122.516,-37.642,179.087,5.489,149.237
C08090=1204.485,-122.267,-37.652,179.089,5.488,149.236
C08091=1204.480,-122.017,-37.661,179.092,5.489,149.235
C08092=1204.474,-121.767,-37.671,179.093,5.489,149.235
C08093=1204.468,-121.517,-37.679,179.095,5.488,149.234
C08094=1204.464,-121.268,-37.689,179.098,5.489,149.233
C08095=1204.458,-121.018,-37.699,179.100,5.489,149.233
C08096=1204.453,-120.769,-37.708,179.102,5.489,149.232
C08097=1204.448,-120.519,-37.717,179.104,5.489,149.231
C08098=1204.442,-120.268,-37.727,179.107,5.489,149.231
C08099=1204.437,-120.019,-37.736,179.109,5.489,149.230
C08100=1204.431,-119.769,-37.746,179.111,5.489,149.229
C08101=1204.426,-119.519,-37.755,179.113,5.489,149.229
C08102=1204.422,-119.269,-37.764,179.116,5.490,149.228
C08103=1204.416,-119.019,-37.774,179.118,5.489,149.227
C08104=1204.411,-118.770,-37.784,179.120,5.490,149.227
C08105=1204.406,-118.520,-37.792,179.122,5.490,149.226
C08106=1204.400,-118.270,-37.802,179.125,5.490,149.226
C08107=1204.395,-118.021,-37.812,179.126,5.490,149.225
C08108=1204.389,-117.770,-37.821,179.129,5.491,149.224
C08109=1204.384,-117.521,-37.831,179.131,5.490,149.224
C08110=1204.379,-117.271,-37.840,179.133,5.491,149.223
C08111=1204.373,-117.022,-37.850,179.135,5.491,149.222
C08112=1204.368,-116.772,-37.859,179.137,5.490,149.222
C08113=1204.363,-116.522,-37.869,179.140,5.491,149.221
C08114=1204.357,-116.273,-37.878,179.142,5.491,149.221
C08115=1204.352,-116.022,-37.888,179.144,5.491,149.220
C08116=1204.347,-115.773,-37.897,179.146,5.491,149.219
C08117=1204.342,-115.523,-37.908,179.149,5.491,149.219
C08118=1204.337,-115.273,-37.916,179.151,5.491,149.218
C08119=1204.332,-115.024,-37.926,179.153,5.492,149.217
C08120=1204.326,-114.774,-37.936,179.155,5.491,149.217
C08121=1204.321,-114.525,-37.945,179.158,5.492,149.216
C08122=1204.315,-114.274,-37.955,179.159,5.492,149.216
C08123=1204.310,-114.025,-37.964,179.162,5.492,149.215
C08124=1204.305,-113.774,-37.974,179.164,5.492,149.214
C08125=1204.300,-113.525,-37.984,179.166,5.493,149.214
C08126=1204.294,-113.275,-37.993,179.168,5.492,149.213
C08127=1204.289,-113.026,-38.003,179.171,5.493,149.212
C08128=1204.283,-112.775,-38.012,179.173,5.492,149.211
C08129=1204.278,-112.526,-38.022,179.175,5.493,149.211
C08130=1204.273,-112.276,-38.031,179.177,5.493,149.210
C08131=1204.268,-112.026,-38.041,179.180,5.493,149.210
C08132=1204.263,-111.777,-38.052,179.182,5.493,149.209
C08133=1204.257,-111.527,-38.060,179.184,5.493,149.208
C08134=1204.252,-111.277,-38.071,179.186,5.493,149.208
C08135=1204.246,-111.027,-38.080,179.189,5.494,149.207
C08136=1204.241,-110.778,-38.090,179.191,5.493,149.206
C08137=1204.236,-110.528,-38.100,179.193,5.494,149.206
C08138=1204.231,-110.278,-38.109,179.195,5.494,149.205
C08139=1204.225,-110.028,-38.119,179.198,5.494,149.204
C08140=1204.221,-109.779,-38.129,179.200,5.494,149.204
C08141=1204.215,-109.529,-38.139,179.202,5.494,149.203
C08142=1204.210,-109.280,-38.148,179.204,5.494,149.203
C08143=1204.205,-109.029,-38.159,179.207,5.495,149.202
C08144=1204.199,-108.779,-38.168,179.209,5.494,149.201
C08145=1204.194,-108.530,-38.178,179.211,5.495,149.201
C08146=1204.188,-108.280,-38.188,179.213,5.495,149.200
C08147=1204.183,-108.031,-38.197,179.216,5.495,149.199
C08148=1204.178,-107.780,-38.208,179.218,5.495,149.199
C08149=1204.173,-107.531,-38.218,179.220,5.496,149.198
C08150=1204.167,-107.281,-38.227,179.222,5.495,149.197
C08151=1204.162,-107.031,-38.237,179.225,5.496,149.197
C08152=1204.157,-106.782,-38.247,179.226,5.496,149.196
C08153=1204.152,-106.532,-38.257,179.229,5.496,149.195
C08154=1204.146,-106.282,-38.267,179.231,5.496,149.195
C08155=1204.141,-106.032,-38.276,179.234,5.496,149.194
C08156=1204.136,-105.783,-38.286,179.235,5.496,149.194
C08157=1204.131,-105.533,-38.297,179.238,5.496,149.193
C08158=1204.125,-105.283,-38.306,179.240,5.496,149.192
C08159=1204.120,-105.033,-38.316,179.242,5.497,149.192
C08160=1204.115,-104.784,-38.326,179.244,5.496,149.191
C08161=1204.110,-104.534,-38.336,179.247,5.497,149.190
C08162=1204.104,-104.284,-38.346,179.249,5.496,149.189
C08163=1204.099,-104.034,-38.355,179.251,5.497,149.189
C08164=1204.094,-103.785,-38.366,179.253,5.497,149.188
C08165=1204.089,-103.535,-38.376,179.256,5.497,149.188
C08166=1204.083,-103.285,-38.386,179.258,5.497,149.187
C08167=1204.078,-103.036,-38.396,179.260,5.498,149.186
C08168=1204.072,-102.786,-38.405,179.263,5.497,149.186
C08169=1204.067,-102.535,-38.416,179.265,5.498,149.185
C08170=1204.062,-102.286,-38.426,179.267,5.498,149.184
C08171=1204.057,-102.037,-38.436,179.269,5.498,149.184
C08172=1204.052,-101.786,-38.446,179.272,5.498,149.183
C08173=1204.046,-101.516,-38.457,179.274,5.498,149.182
C08174=1204.041,-101.244,-38.467,179.276,5.498,149.182
C08175=1204.035,-100.972,-38.479,179.279,5.498,149.181
C08176=1204.029,-100.702,-38.489,179.282,5.499,149.180
C08177=1204.024,-100.451,-38.500,179.283,5.499,149.180
C08178=1204.018,-100.202,-38.510,179.286,5.499,149.179
C08179=1204.013,-99.953,-38.520,179.288,5.499,149.178
C08180=1204.008,-99.702,-38.530,179.291,5.499,149.178
C08181=1204.002,-99.452,-38.540,179.292,5.499,149.177
C08182=1203.997,-99.203,-38.550,179.295,5.499,149.176
C08183=1203.992,-98.952,-38.561,179.297,5.499,149.176
C08184=1203.987,-98.703,-38.570,179.300,5.500,149.175
C08185=1203.981,-98.454,-38.580,179.301,5.500,149.174
C08186=1203.976,-98.203,-38.591,179.304,5.500,149.174
C08187=1203.971,-97.954,-38.601,179.306,5.500,149.173
C08188=1203.966,-97.705,-38.611,179.309,5.500,149.172
C08189=1203.961,-97.454,-38.621,179.311,5.501,149.172
C08190=1203.955,-97.205,-38.632,179.313,5.500,149.171
C08191=1203.950,-96.955,-38.642,179.316,5.501,149.170
C08192=1203.945,-96.705,-38.652,179.318,5.500,149.170
C08193=1203.939,-96.456,-38.663,179.320,5.501,149.169
C08194=1203.934,-96.206,-38.672,179.322,5.501,149.168
C08195=1203.929,-95.956,-38.683,179.325,5.501,149.168
C08196=1203.924,-95.707,-38.693,179.327,5.501,149.167
C08197=1203.918,-95.457,-38.703,179.329,5.502,149.167
C08198=1203.913,-95.207,-38.714,179.331,5.501,149.166
C08199=1203.908,-94.957,-38.724,179.334,5.502,149.165
C08200=1203.903,-94.707,-38.734,179.336,5.501,149.164
C08201=1203.898,-94.458,-38.744,179.338,5.502,149.164
C08202=1203.892,-94.208,-38.754,179.340,5.502,149.163
C08203=1203.887,-93.958,-38.765,179.343,5.502,149.163
C08204=1203.881,-93.708,-38.775,179.345,5.502,149.162
C08205=1203.877,-93.459,-38.786,179.347,5.503,149.161
C08206=1203.871,-93.209,-38.797,179.350,5.503,149.161
C08207=1203.866,-92.960,-38.807,179.352,5.503,149.160
C08208=1203.861,-92.710,-38.817,179.355,5.503,149.159
C08209=1203.856,-92.460,-38.827,179.356,5.503,149.159
C08210=1203.851,-92.210,-38.838,179.359,5.503,149.158
C08211=1203.845,-91.960,-38.848,179.361,5.503,149.157
C08212=1203.840,-91.711,-38.858,179.364,5.504,149.157
C08213=1203.835,-91.461,-38.869,179.365,5.504,149.156
C08214=1203.829,-91.212,-38.880,179.368,5.504,149.155
C08215=1203.824,-90.961,-38.890,179.370,5.504,149.155
C08216=1203.819,-90.712,-38.900,179.373,5.504,149.154
C08217=1203.813,-90.462,-38.911,179.374,5.504,149.153
C08218=1203.808,-90.212,-38.921,179.377,5.504,149.153
C08219=1203.802,-89.963,-38.931,179.380,5.505,149.152
C08220=1203.798,-89.713,-38.943,179.382,5.504,149.151
C08221=1203.793,-89.464,-38.952,179.384,5.505,149.151
C08222=1203.788,-89.213,-38.963,179.386,5.505,149.150
C08223=1203.782,-88.964,-38.973,179.389,5.505,149.149
C08224=1203.777,-88.714,-38.984,179.391,5.505,149.149
C08225=1203.772,-88.465,-38.995,179.393,5.505,149.148
C08226=1203.767,-88.215,-39.005,179.395,5.505,149.148
C08227=1203.761,-87.965,-39.015,179.398,5.506,149.147
C08228=1203.756,-87.715,-39.025,179.400,5.505,149.146
C08229=1203.751,-87.466,-39.037,179.402,5.506,149.145
C08230=1203.746,-87.216,-39.047,179.405,5.507,149.145
C08231=1203.741,-86.966,-39.058,179.407,5.506,149.144
C08232=1203.735,-86.716,-39.068,179.409,5.507,149.144
C08233=1203.730,-86.467,-39.079,179.411,5.506,149.143
C08234=1203.725,-86.217,-39.089,179.414,5.507,149.142
C08235=1203.720,-85.967,-39.100,179.416,5.507,149.142
C08236=1203.714,-85.718,-39.110,179.418,5.507,149.141
C08237=1203.709,-85.468,-39.121,179.420,5.507,149.140
C08238=1203.704,-85.218,-39.132,179.423,5.507,149.139
C08239=1203.699,-84.968,-39.142,179.426,5.508,149.139
C08240=1203.693,-84.719,-39.154,179.427,5.508,149.138
C08241=1203.688,-84.469,-39.164,179.430,5.508,149.138
C08242=1203.682,-84.219,-39.174,179.432,5.508,149.137
C08243=1203.677,-83.969,-39.186,179.435,5.508,149.136
C08244=1203.672,-83.719,-39.196,179.436,5.508,149.136
C08245=1203.667,-83.470,-39.207,179.439,5.509,149.135
C08246=1203.662,-83.220,-39.218,179.441,5.508,149.134
C08247=1203.657,-82.971,-39.228,179.444,5.509,149.134
C08248=1203.652,-82.721,-39.239,179.447,5.509,149.133
C08249=1203.646,-82.471,-39.250,179.448,5.509,149.132
C08250=1203.641,-82.221,-39.260,179.451,5.510,149.132
C08251=1203.636,-81.972,-39.271,179.453,5.509,149.131
C08252=1203.631,-81.722,-39.282,179.456,5.510,149.130
C08253=1203.625,-81.473,-39.293,179.458,5.509,149.130
C08254=1203.620,-81.222,-39.304,179.460,5.510,149.129
C08255=1203.615,-80.972,-39.314,179.462,5.510,149.128
C08256=1203.610,-80.723,-39.325,179.465,5.510,149.128
C08257=1203.605,-80.473,-39.336,179.467,5.511,149.127
C08258=1203.599,-80.224,-39.347,179.469,5.511,149.126
C08259=1203.594,-79.974,-39.357,179.472,5.511,149.126
C08260=1203.588,-79.725,-39.369,179.474,5.511,149.125
C08261=1203.583,-79.474,-39.379,179.476,5.511,149.124
C08262=1203.579,-79.225,-39.391,179.479,5.511,149.124
C08263=1203.573,-78.975,-39.401,179.481,5.511,149.123
C08264=1203.568,-78.726,-39.412,179.483,5.512,149.122
C08265=1203.563,-78.476,-39.422,179.485,5.512,149.122
C08266=1203.557,-78.226,-39.434,179.488,5.512,149.121
C08267=1203.552,-77.976,-39.445,179.490,5.512,149.120
C08268=1203.547,-77.727,-39.456,179.492,5.512,149.120
C08269=1203.542,-77.477,-39.466,179.495,5.513,149.119
C08270=1203.537,-77.228,-39.477,179.497,5.512,149.118
C08271=1203.531,-76.977,-39.488,179.500,5.513,149.118
C08272=1203.526,-76.728,-39.500,179.502,5.513,149.117
C08273=1203.521,-76.478,-39.510,179.504,5.513,149.116
C08274=1203.516,-76.228,-39.521,179.506,5.513,149.116
C08275=1203.510,-75.979,-39.531,179.509,5.513,149.115
C08276=1203.505,-75.729,-39.543,179.511,5.514,149.114
C08277=1203.500,-75.458,-39.555,179.513,5.513,149.114
C08278=1203.494,-75.188,-39.567,179.516,5.514,149.113
C08279=1203.488,-74.917,-39.579,179.519,5.514,149.112
C08280=1203.483,-74.646,-39.591,179.521,5.514,149.112
C08281=1203.477,-74.396,-39.602,179.524,5.514,149.111
C08282=1203.472,-74.147,-39.613,179.526,5.515,149.110
C08283=1203.467,-73.897,-39.625,179.528,5.515,149.110
C08284=1203.461,-73.647,-39.635,179.530,5.515,149.109
C08285=1203.457,-73.398,-39.646,179.533,5.515,149.108
C08286=1203.451,-73.148,-39.656,179.535,5.515,149.107
C08287=1203.446,-72.898,-39.668,179.538,5.516,149.107
C08288=1203.441,-72.649,-39.680,179.540,5.515,149.106
C08289=1203.435,-72.399,-39.690,179.542,5.516,149.106
C08290=1203.430,-72.149,-39.702,179.544,5.516,149.105
C08291=1203.425,-71.900,-39.713,179.547,5.516,149.104
C08292=1203.420,-71.649,-39.724,179.550,5.517,149.103
C08293=1203.414,-71.400,-39.735,179.552,5.516,149.103
C08294=1203.410,-71.150,-39.746,179.554,5.517,149.102
C08295=1203.405,-70.901,-39.758,179.556,5.517,149.102
C08296=1203.398,-70.651,-39.768,179.559,5.517,149.101
C08297=1203.394,-70.401,-39.780,179.561,5.518,149.100
C08298=1203.389,-70.152,-39.791,179.563,5.517,149.099
C08299=1203.383,-69.902,-39.802,179.566,5.518,149.099
C08300=1203.378,-69.652,-39.813,179.568,5.518,149.098
C08301=1203.373,-69.403,-39.824,179.570,5.518,149.098
C08302=1203.368,-69.153,-39.836,179.573,5.519,149.097
C08303=1203.362,-68.903,-39.847,179.575,5.518,149.096
C08304=1203.358,-68.654,-39.858,179.578,5.519,149.095
C08305=1203.352,-68.404,-39.870,179.579,5.519,149.095
C08306=1203.347,-68.155,-39.881,179.582,5.519,149.094
C08307=1203.342,-67.905,-39.892,179.585,5.520,149.094
C08308=1203.337,-67.654,-39.903,179.587,5.519,149.093
C08309=1203.332,-67.405,-39.914,179.589,5.520,149.092
C08310=1203.326,-67.156,-39.926,179.591,5.520,149.092
C08311=1203.321,-66.906,-39.937,179.594,5.520,149.091
C08312=1203.316,-66.656,-39.949,179.596,5.521,149.090
C08313=1203.311,-66.406,-39.960,179.598,5.520,149.090
C08314=1203.305,-66.157,-39.971,179.601,5.521,149.089
C08315=1203.300,-65.907,-39.982,179.603,5.520,149.088
C08316=1203.295,-65.657,-39.994,179.605,5.521,149.088
C08317=1203.290,-65.407,-40.006,179.608,5.522,149.087
C08318=1203.285,-65.158,-40.017,179.610,5.521,149.086
C08319=1203.279,-64.909,-40.028,179.613,5.522,149.086
C08320=1203.274,-64.659,-40.040,179.615,5.522,149.085
C08321=1203.269,-64.408,-40.051,179.618,5.522,149.084
C08322=1203.264,-64.159,-40.062,179.620,5.523,149.084
C08323=1203.258,-63.909,-40.074,179.622,5.522,149.083
C08324=1203.253,-63.660,-40.085,179.624,5.523,149.082
C08325=1203.249,-63.410,-40.096,179.627,5.523,149.082
C08326=1203.243,-63.160,-40.108,179.629,5.523,149.081
C08327=1203.238,-62.911,-40.119,179.631,5.524,149.080
C08328=1203.232,-62.661,-40.131,179.634,5.524,149.080
C08329=1203.228,-62.412,-40.142,179.636,5.524,149.079
C08330=1203.222,-62.162,-40.154,179.639,5.524,149.078
C08331=1203.218,-61.912,-40.165,179.641,5.524,149.078
C08332=1203.212,-61.662,-40.177,179.644,5.524,149.077
C08333=1203.207,-61.413,-40.189,179.646,5.525,149.076
C08334=1203.201,-61.163,-40.200,179.648,5.525,149.076
C08335=1203.196,-60.914,-40.212,179.651,5.525,149.075
C08336=1203.191,-60.664,-40.223,179.653,5.526,149.074
C08337=1203.186,-60.414,-40.235,179.655,5.525,149.074
C08338=1203.181,-60.164,-40.246,179.658,5.526,149.073
C08339=1203.176,-59.914,-40.258,179.660,5.526,149.072
C08340=1203.171,-59.665,-40.269,179.662,5.526,149.072
C08341=1203.165,-59.416,-40.281,179.665,5.527,149.071
C08342=1203.160,-59.166,-40.292,179.667,5.526,149.070
C08343=1203.155,-58.916,-40.304,179.670,5.527,149.070
C08344=1203.150,-58.666,-40.316,179.672,5.527,149.069
C08345=1203.145,-58.416,-40.328,179.674,5.527,149.068
C08346=1203.139,-58.166,-40.339,179.677,5.528,149.068
C08347=1203.135,-57.917,-40.351,179.679,5.528,149.067
C08348=1203.129,-57.668,-40.362,179.681,5.528,149.066
C08349=1203.124,-57.418,-40.373,179.684,5.528,149.066
C08350=1203.119,-57.168,-40.385,179.686,5.528,149.065
C08351=1203.113,-56.919,-40.398,179.688,5.529,149.064
C08352=1203.109,-56.669,-40.409,179.691,5.529,149.064
C08353=1203.103,-56.419,-40.421,179.693,5.529,149.063
C08354=1203.098,-56.169,-40.433,179.696,5.529,149.062
C08355=1203.093,-55.920,-40.444,179.698,5.530,149.062
C08356=1203.088,-55.670,-40.456,179.700,5.529,149.061
C08357=1203.083,-55.420,-40.468,179.703,5.530,149.060
C08358=1203.077,-55.171,-40.480,179.705,5.530,149.060
C08359=1203.072,-54.921,-40.492,179.707,5.530,149.059
C08360=1203.067,-54.672,-40.503,179.710,5.531,149.058
C08361=1203.062,-54.422,-40.515,179.713,5.531,149.058
C08362=1203.056,-54.172,-40.527,179.715,5.531,149.057
C08363=1203.052,-53.923,-40.539,179.717,5.531,149.056
C08364=1203.047,-53.673,-40.551,179.720,5.532,149.056
C08365=1203.041,-53.423,-40.562,179.722,5.532,149.055
C08366=1203.036,-53.173,-40.574,179.724,5.532,149.054
C08367=1203.031,-52.924,-40.586,179.727,5.532,149.054
C08368=1203.026,-52.674,-40.598,179.729,5.532,149.053
C08369=1203.021,-52.425,-40.610,179.732,5.533,149.052
C08370=1203.016,-52.175,-40.621,179.733,5.533,149.052
C08371=1203.010,-51.925,-40.633,179.736,5.533,149.051
C08372=1203.005,-51.675,-40.646,179.739,5.534,149.050
C08373=1203.001,-51.426,-40.657,179.741,5.533,149.050
C08374=1202.995,-51.176,-40.669,179.743,5.534,149.049
C08375=1202.990,-50.926,-40.681,179.746,5.534,149.048
C08376=1202.985,-50.677,-40.694,179.748,5.534,149.047
C08377=1202.980,-50.427,-40.705,179.750,5.535,149.047
C08378=1202.974,-50.177,-40.717,179.753,5.535,149.046
C08379=1202.969,-49.928,-40.729,179.755,5.535,149.046
C08380=1202.964,-49.678,-40.741,179.758,5.535,149.045
C08381=1202.958,-49.408,-40.754,179.760,5.536,149.044
C08382=1202.953,-49.138,-40.767,179.763,5.536,149.043
C08383=1202.947,-48.868,-40.779,179.766,5.536,149.043
C08384=1202.941,-48.598,-40.792,179.768,5.536,149.042
C08385=1202.936,-48.348,-40.805,179.771,5.537,149.041
C08386=1202.931,-48.099,-40.817,179.773,5.537,149.041
C08387=1202.925,-47.849,-40.829,179.775,5.537,149.040
C08388=1202.921,-47.600,-40.841,179.778,5.537,149.039
C08389=1202.916,-47.350,-40.853,179.780,5.538,149.039
C08390=1202.910,-47.100,-40.865,179.782,5.538,149.038
C08391=1202.905,-46.850,-40.877,179.785,5.538,149.037
C08392=1202.900,-46.600,-40.889,179.788,5.539,149.037
C08393=1202.895,-46.351,-40.901,179.790,5.538,149.036
C08394=1202.890,-46.101,-40.913,179.792,5.539,149.035
C08395=1202.885,-45.852,-40.925,179.795,5.539,149.035
C08396=1202.879,-45.602,-40.937,179.797,5.539,149.034
C08397=1202.874,-45.353,-40.950,179.799,5.540,149.033
C08398=1202.869,-45.102,-40.962,179.802,5.540,149.033
C08399=1202.864,-44.852,-40.974,179.805,5.540,149.032
C08400=1202.859,-44.603,-40.987,179.807,5.540,149.031
C08401=1202.854,-44.353,-40.998,179.809,5.541,149.031
C08402=1202.849,-44.104,-41.011,179.811,5.541,149.030
C08403=1202.844,-43.854,-41.022,179.814,5.541,149.029
C08404=1202.838,-43.605,-41.035,179.816,5.542,149.029
C08405=1202.833,-43.355,-41.047,179.819,5.542,149.028
C08406=1202.828,-43.106,-41.060,179.821,5.542,149.027
C08407=1202.822,-42.856,-41.071,179.824,5.542,149.027
C08408=1202.817,-42.606,-41.084,179.826,5.543,149.026
C08409=1202.812,-42.357,-41.097,179.828,5.543,149.025
C08410=1202.807,-42.107,-41.109,179.831,5.543,149.025
C08411=1202.803,-41.857,-41.121,179.833,5.544,149.024
C08412=1202.798,-41.607,-41.133,179.835,5.543,149.023
C08413=1202.792,-41.358,-41.145,179.838,5.544,149.023
C08414=1202.787,-41.108,-41.157,179.841,5.544,149.022
C08415=1202.782,-40.859,-41.170,179.843,5.545,149.021
C08416=1202.776,-40.609,-41.182,179.845,5.545,149.021
C08417=1202.771,-40.360,-41.194,179.848,5.545,149.020
C08418=1202.766,-40.110,-41.207,179.850,5.546,149.019
C08419=1202.761,-39.860,-41.219,179.852,5.545,149.019
C08420=1202.756,-39.610,-41.232,179.855,5.546,149.018
C08421=1202.751,-39.361,-41.244,179.858,5.546,149.017
C08422=1202.746,-39.111,-41.256,179.860,5.547,149.017
C08423=1202.741,-38.862,-41.269,179.862,5.547,149.016
C08424=1202.735,-38.612,-41.281,179.864,5.547,149.015
C08425=1202.730,-38.362,-41.293,179.867,5.548,149.015
C08426=1202.725,-38.113,-41.306,179.869,5.547,149.014
C08427=1202.720,-37.863,-41.318,179.872,5.548,149.013
C08428=1202.715,-37.613,-41.331,179.875,5.548,149.013
C08429=1202.710,-37.364,-41.343,179.877,5.548,149.012
C08430=1202.704,-37.114,-41.355,179.879,5.549,149.011
C08431=1202.699,-36.865,-41.368,179.881,5.549,149.011
C08432=1202.694,-36.615,-41.381,179.884,5.550,149.010
C08433=1202.690,-36.365,-41.393,179.886,5.549,149.009
C08434=1202.684,-36.115,-41.405,179.889,5.550,149.009
C08435=1202.679,-35.866,-41.418,179.892,5.550,149.008
C08436=1202.673,-35.616,-41.431,179.893,5.550,149.007
C08437=1202.668,-35.367,-41.444,179.896,5.551,149.007
C08438=1202.663,-35.116,-41.456,179.898,5.551,149.006
C08439=1202.658,-34.867,-41.469,179.901,5.552,149.005
C08440=1202.653,-34.618,-41.481,179.903,5.551,149.005
C08441=1202.648,-34.369,-41.494,179.906,5.552,149.004
C08442=1202.642,-34.119,-41.506,179.909,5.552,149.003
C08443=1202.638,-33.869,-41.519,179.911,5.553,149.003
C08444=1202.633,-33.619,-41.531,179.913,5.553,149.002
C08445=1202.628,-33.370,-41.544,179.915,5.553,149.001
C08446=1202.622,-33.120,-41.557,179.918,5.554,149.001
C08447=1202.616,-32.870,-41.569,179.920,5.553,149.000
C08448=1202.612,-32.620,-41.582,179.923,5.554,148.999
C08449=1202.607,-32.371,-41.595,179.926,5.554,148.999
C08450=1202.602,-32.122,-41.607,179.928,5.555,148.998
C08451=1202.596,-31.872,-41.620,179.930,5.555,148.997
C08452=1202.592,-31.622,-41.633,179.932,5.555,148.997
C08453=1202.586,-31.372,-41.645,179.935,5.556,148.996
C08454=1202.581,-31.123,-41.658,179.938,5.556,148.995
C08455=1202.576,-30.873,-41.670,179.940,5.556,148.995
C08456=1202.571,-30.623,-41.683,179.942,5.556,148.994
C08457=1202.566,-30.374,-41.696,179.945,5.557,148.993
C08458=1202.561,-30.125,-41.709,179.947,5.558,148.993
C08459=1202.555,-29.875,-41.722,179.949,5.557,148.992
C08460=1202.550,-29.625,-41.735,179.952,5.558,148.991
C08461=1202.545,-29.376,-41.747,179.955,5.558,148.991
C08462=1202.540,-29.127,-41.760,179.957,5.559,148.990
C08463=1202.536,-28.877,-41.773,179.959,5.558,148.989
C08464=1202.529,-28.626,-41.785,179.962,5.559,148.989
C08465=1202.524,-28.377,-41.798,179.964,5.560,148.988
C08466=1202.519,-28.128,-41.811,179.966,5.559,148.987
C08467=1202.515,-27.878,-41.824,179.969,5.560,148.987
C08468=1202.509,-27.628,-41.837,179.972,5.560,148.986
C08469=1202.504,-27.379,-41.849,179.974,5.561,148.985
C08470=1202.499,-27.129,-41.862,179.976,5.560,148.985
C08471=1202.494,-26.879,-41.875,179.979,5.561,148.984
C08472=1202.489,-26.630,-41.887,179.981,5.562,148.983
C08473=1202.484,-26.380,-41.901,179.984,5.562,148.983
C08474=1202.479,-26.130,-41.914,179.987,5.563,148.982
C08475=1202.473,-25.881,-41.926,179.989,5.562,148.981
C08476=1202.468,-25.631,-41.940,179.991,5.563,148.981
C08477=1202.463,-25.381,-41.952,179.994,5.563,148.980
C08478=1202.458,-25.133,-41.966,179.996,5.564,148.979
C08479=1202.454,-24.883,-41.979,179.998,5.564,148.979
C08480=1202.448,-24.633,-41.992,-179.999,5.564,148.978
C08481=1202.443,-24.384,-42.005,-179.996,5.565,148.977
C08482=1202.438,-24.134,-42.017,-179.994,5.565,148.977
C08483=1202.432,-23.884,-42.031,-179.992,5.565,148.976
C08484=1202.427,-23.635,-42.043,-179.989,5.565,148.975
C08485=1202.422,-23.365,-42.057,-179.986,5.566,148.975
C08486=1202.417,-23.096,-42.072,-179.984,5.566,148.974
C08487=1202.411,-22.826,-42.086,-179.981,5.567,148.973
C08488=1202.405,-22.557,-42.100,-179.978,5.567,148.973
C08489=1202.400,-22.306,-42.113,-179.976,5.568,148.972
C08490=1202.395,-22.057,-42.126,-179.974,5.567,148.971
C08491=1202.390,-21.808,-42.138,-179.971,5.568,148.971
C08492=1202.385,-21.558,-42.153,-179.969,5.569,148.970
C08493=1202.380,-21.309,-42.165,-179.966,5.569,148.969
C08494=1202.375,-21.059,-42.178,-179.964,5.569,148.969
C08495=1202.369,-20.809,-42.191,-179.961,5.569,148.968
C08496=1202.364,-20.560,-42.204,-179.959,5.570,148.967
C08497=1202.359,-20.310,-42.218,-179.956,5.570,148.966
C08498=1202.354,-20.061,-42.231,-179.954,5.571,148.966
C08499=1202.350,-19.811,-42.244,-179.952,5.571,148.965
C08500=1202.344,-19.561,-42.257,-179.949,5.571,148.965
C08501=1202.339,-19.312,-42.270,-179.947,5.572,148.964
C08502=1202.334,-19.062,-42.284,-179.944,5.572,148.963
C08503=1202.329,-18.813,-42.296,-179.942,5.572,148.963
C08504=1202.323,-18.562,-42.310,-179.939,5.572,148.962
C08505=1202.318,-18.313,-42.323,-179.937,5.573,148.961
C08506=1202.314,-18.064,-42.336,-179.934,5.574,148.961
C08507=1202.308,-17.814,-42.349,-179.932,5.574,148.960
C08508=1202.303,-17.565,-42.362,-179.930,5.574,148.959
C08509=1202.298,-17.315,-42.376,-179.927,5.574,148.959
C08510=1202.293,-17.066,-42.389,-179.924,5.575,148.958
C08511=1202.288,-16.815,-42.403,-179.922,5.575,148.957
C08512=1202.283,-16.566,-42.415,-179.919,5.576,148.957
C08513=1202.278,-16.316,-42.429,-179.917,5.576,148.956
C08514=1202.273,-16.067,-42.442,-179.915,5.576,148.955
C08515=1202.267,-15.817,-42.456,-179.912,5.577,148.955
C08516=1202.262,-15.568,-42.469,-179.909,5.577,148.954
C08517=1202.257,-15.318,-42.482,-179.907,5.578,148.953
C08518=1202.252,-15.069,-42.496,-179.905,5.578,148.953
C08519=1202.247,-14.819,-42.509,-179.903,5.578,148.952
C08520=1202.242,-14.569,-42.522,-179.900,5.579,148.951
C08521=1202.237,-14.320,-42.536,-179.897,5.579,148.951
C08522=1202.232,-14.070,-42.549,-179.895,5.580,148.950
C08523=1202.227,-13.820,-42.563,-179.892,5.579,148.949
C08524=1202.222,-13.571,-42.576,-179.890,5.580,148.949
C08525=1202.217,-13.321,-42.589,-179.888,5.581,148.948
C08526=1202.211,-13.072,-42.603,-179.885,5.581,148.948
C08527=1202.206,-12.822,-42.616,-179.882,5.582,148.947
C08528=1202.201,-12.573,-42.630,-179.880,5.581,148.946
C08529=1202.196,-12.323,-42.643,-179.878,5.582,148.945
C08530=1202.191,-12.074,-42.657,-179.875,5.582,148.945
C08531=1202.186,-11.824,-42.670,-179.872,5.583,148.944
C08532=1202.181,-11.575,-42.684,-179.870,5.584,148.944
C08533=1202.175,-11.324,-42.697,-179.868,5.583,148.943
C08534=1202.170,-11.075,-42.710,-179.865,5.584,148.942
C08535=1202.165,-10.825,-42.724,-179.863,5.584,148.942
C08536=1202.161,-10.576,-42.738,-179.860,5.585,148.941
C08537=1202.155,-10.326,-42.751,-179.857,5.585,148.940
C08538=1202.150,-10.077,-42.765,-179.855,5.586,148.940
C08539=1202.145,-9.827,-42.778,-179.853,5.586,148.939
C08540=1202.140,-9.578,-42.792,-179.851,5.586,148.938
C08541=1202.134,-9.328,-42.805,-179.848,5.587,148.938
C08542=1202.130,-9.079,-42.819,-179.845,5.587,148.937
C08543=1202.125,-8.828,-42.833,-179.843,5.588,148.936
C08544=1202.120,-8.580,-42.846,-179.840,5.587,148.936
C08545=1202.115,-8.329,-42.860,-179.838,5.588,148.935
C08546=1202.109,-8.080,-42.873,-179.836,5.589,148.934
C08547=1202.105,-7.831,-42.887,-179.833,5.589,148.934
C08548=1202.099,-7.581,-42.900,-179.830,5.590,148.933
C08549=1202.094,-7.331,-42.915,-179.828,5.590,148.932
C08550=1202.090,-7.081,-42.928,-179.826,5.590,148.932
C08551=1202.084,-6.832,-42.942,-179.823,5.591,148.931
C08552=1202.079,-6.583,-42.956,-179.821,5.591,148.930
C08553=1202.074,-6.332,-42.969,-179.818,5.592,148.930
C08554=1202.069,-6.084,-42.983,-179.815,5.592,148.929
C08555=1202.064,-5.834,-42.997,-179.813,5.593,148.928
C08556=1202.058,-5.584,-43.010,-179.810,5.593,148.928
C08557=1202.054,-5.335,-43.024,-179.808,5.593,148.927
C08558=1202.049,-5.085,-43.038,-179.806,5.594,148.927
C08559=1202.043,-4.836,-43.051,-179.803,5.594,148.926
C08560=1202.038,-4.586,-43.066,-179.801,5.595,148.925
C08561=1202.034,-4.337,-43.079,-179.798,5.595,148.924
C08562=1202.028,-4.087,-43.092,-179.795,5.596,148.924
C08563=1202.023,-3.837,-43.107,-179.793,5.595,148.923
C08564=1202.018,-3.587,-43.121,-179.791,5.596,148.923
C08565=1202.013,-3.338,-43.135,-179.788,5.597,148.922
C08566=1202.008,-3.088,-43.148,-179.786,5.597,148.921
C08567=1202.003,-2.839,-43.162,-179.783,5.598,148.921
C08568=1201.998,-2.590,-43.176,-179.780,5.598,148.920
C08569=1201.993,-2.340,-43.190,-179.778,5.599,148.919
C08570=1201.988,-2.090,-43.203,-179.776,5.599,148.919
C08571=1201.983,-1.841,-43.217,-179.774,5.599,148.918
C08572=1201.978,-1.591,-43.232,-179.771,5.600,148.917
C08573=1201.973,-1.342,-43.246,-179.768,5.600,148.917
C08574=1201.967,-1.093,-43.260,-179.766,5.601,148.916
C08575=1201.962,-0.842,-43.273,-179.763,5.601,148.915
C08576=1201.958,-0.593,-43.287,-179.760,5.602,148.915
C08577=1201.952,-0.344,-43.301,-179.759,5.602,148.914
C08578=1201.947,-0.094,-43.315,-179.756,5.602,148.913
C08579=1201.942,0.156,-43.329,-179.753,5.603,148.913
C08580=1201.937,0.405,-43.344,-179.751,5.603,148.912
C08581=1201.932,0.655,-43.357,-179.748,5.604,148.911
C08582=1201.927,0.905,-43.371,-179.745,5.604,148.911
C08583=1201.922,1.154,-43.385,-179.743,5.605,148.910
C08584=1201.917,1.403,-43.399,-179.741,5.606,148.910
C08585=1201.912,1.653,-43.413,-179.739,5.605,148.909
C08586=1201.907,1.902,-43.427,-179.736,5.606,148.908
C08587=1201.902,2.152,-43.442,-179.733,5.606,148.907
C08588=1201.896,2.401,-43.456,-179.731,5.607,148.907
C08589=1201.891,2.671,-43.470,-179.728,5.607,148.906
C08590=1201.886,2.940,-43.485,-179.725,5.608,148.905
C08591=1201.880,3.209,-43.501,-179.723,5.608,148.905
C08592=1201.875,3.478,-43.516,-179.720,5.609,148.904
C08593=1201.869,3.727,-43.530,-179.717,5.609,148.903
C08594=1201.864,3.977,-43.544,-179.715,5.610,148.903
C08595=1201.860,4.227,-43.559,-179.712,5.611,148.902
C08596=1201.855,4.476,-43.573,-179.710,5.611,148.901
C08597=1201.850,4.726,-43.587,-179.707,5.612,148.901
C08598=1201.844,4.975,-43.601,-179.705,5.611,148.900
C08599=1201.839,5.225,-43.615,-179.702,5.612,148.899
C08600=1201.834,5.475,-43.630,-179.700,5.613,148.899
C08601=1201.829,5.724,-43.644,-179.698,5.613,148.898
C08602=1201.824,5.974,-43.658,-179.695,5.614,148.898
C08603=1201.819,6.223,-43.672,-179.692,5.614,148.897
C08604=1201.814,6.473,-43.686,-179.690,5.615,148.896
C08605=1201.809,6.722,-43.701,-179.687,5.615,148.896
C08606=1201.804,6.972,-43.715,-179.685,5.616,148.895
C08607=1201.799,7.222,-43.729,-179.683,5.616,148.894
C08608=1201.794,7.470,-43.744,-179.680,5.616,148.894
C08609=1201.789,7.720,-43.758,-179.677,5.617,148.893
C08610=1201.784,7.970,-43.772,-179.675,5.617,148.892
C08611=1201.779,8.219,-43.787,-179.672,5.618,148.892
C08612=1201.774,8.469,-43.801,-179.670,5.619,148.891
C08613=1201.769,8.719,-43.815,-179.667,5.619,148.891
C08614=1201.763,8.968,-43.829,-179.665,5.620,148.890
C08615=1201.758,9.217,-43.843,-179.662,5.620,148.889
C08616=1201.753,9.467,-43.858,-179.659,5.621,148.888
C08617=1201.749,9.716,-43.873,-179.657,5.622,148.888
C08618=1201.744,9.966,-43.887,-179.655,5.621,148.887
C08619=1201.739,10.216,-43.901,-179.653,5.622,148.887
C08620=1201.734,10.465,-43.916,-179.650,5.622,148.886
C08621=1201.728,10.714,-43.929,-179.647,5.623,148.885
C08622=1201.723,10.964,-43.945,-179.645,5.623,148.885
C08623=1201.718,11.214,-43.959,-179.642,5.624,148.884
C08624=1201.713,11.463,-43.974,-179.640,5.625,148.883
C08625=1201.708,11.713,-43.988,-179.637,5.625,148.883
C08626=1201.703,11.963,-44.002,-179.634,5.626,148.882
C08627=1201.698,12.212,-44.017,-179.632,5.626,148.881
C08628=1201.693,12.461,-44.031,-179.630,5.627,148.881
C08629=1201.689,12.711,-44.046,-179.627,5.627,148.880
C08630=1201.682,12.960,-44.060,-179.625,5.627,148.880
C08631=1201.678,13.210,-44.075,-179.622,5.628,148.879
C08632=1201.673,13.459,-44.089,-179.620,5.628,148.878
C08633=1201.668,13.709,-44.104,-179.617,5.629,148.878
C08634=1201.663,13.958,-44.119,-179.615,5.630,148.877
C08635=1201.658,14.208,-44.133,-179.612,5.630,148.876
C08636=1201.652,14.458,-44.148,-179.610,5.631,148.876
C08637=1201.647,14.708,-44.162,-179.607,5.631,148.875
C08638=1201.643,14.957,-44.177,-179.604,5.632,148.874
C08639=1201.638,15.206,-44.191,-179.602,5.632,148.874
C08640=1201.633,15.456,-44.206,-179.599,5.633,148.873
C08641=1201.627,15.705,-44.221,-179.597,5.633,148.872
C08642=1201.623,15.955,-44.236,-179.594,5.634,148.872
C08643=1201.618,16.204,-44.251,-179.591,5.634,148.871
C08644=1201.612,16.453,-44.264,-179.589,5.635,148.870
C08645=1201.607,16.703,-44.279,-179.587,5.635,148.870
C08646=1201.602,16.952,-44.294,-179.585,5.636,148.869
C08647=1201.597,17.202,-44.309,-179.582,5.636,148.869
C08648=1201.592,17.451,-44.324,-179.579,5.637,148.868
C08649=1201.587,17.701,-44.338,-179.577,5.637,148.867
C08650=1201.582,17.951,-44.353,-179.575,5.638,148.867
C08651=1201.577,18.200,-44.368,-179.572,5.638,148.866
C08652=1201.572,18.450,-44.382,-179.569,5.639,148.865
C08653=1201.567,18.699,-44.398,-179.567,5.640,148.865
C08654=1201.562,18.949,-44.412,-179.564,5.640,148.864
C08655=1201.557,19.198,-44.427,-179.562,5.641,148.864
C08656=1201.552,19.448,-44.441,-179.559,5.641,148.863
C08657=1201.547,19.697,-44.457,-179.556,5.642,148.862
C08658=1201.542,19.947,-44.471,-179.554,5.642,148.862
C08659=1201.537,20.196,-44.486,-179.551,5.643,148.861
C08660=1201.531,20.446,-44.501,-179.549,5.644,148.860
C08661=1201.527,20.695,-44.516,-179.546,5.644,148.860
C08662=1201.522,20.945,-44.530,-179.544,5.645,148.859
C08663=1201.516,21.194,-44.546,-179.541,5.645,148.858
C08664=1201.512,21.444,-44.560,-179.538,5.646,148.858
C08665=1201.507,21.693,-44.575,-179.536,5.647,148.857
C08666=1201.502,21.944,-44.590,-179.534,5.647,148.857
C08667=1201.497,22.193,-44.605,-179.531,5.648,148.856
C08668=1201.492,22.442,-44.620,-179.529,5.647,148.855
C08669=1201.487,22.692,-44.635,-179.526,5.648,148.855
C08670=1201.482,22.941,-44.650,-179.524,5.649,148.854
C08671=1201.476,23.191,-44.665,-179.521,5.649,148.853
C08672=1201.472,23.440,-44.680,-179.519,5.650,148.853
C08673=1201.467,23.690,-44.694,-179.516,5.650,148.852
C08674=1201.461,23.939,-44.710,-179.514,5.651,148.851
C08675=1201.457,24.188,-44.725,-179.511,5.652,148.851
C08676=1201.451,24.438,-44.740,-179.509,5.652,148.850
C08677=1201.446,24.687,-44.755,-179.506,5.653,148.850
C08678=1201.442,24.936,-44.770,-179.503,5.653,148.849
C08679=1201.436,25.186,-44.785,-179.501,5.654,148.848
C08680=1201.432,25.436,-44.800,-179.499,5.655,148.848
C08681=1201.427,25.686,-44.816,-179.496,5.655,148.847
C08682=1201.422,25.935,-44.830,-179.493,5.656,148.846
C08683=1201.416,26.185,-44.845,-179.491,5.656,148.846
C08684=1201.412,26.434,-44.860,-179.489,5.657,148.845
C08685=1201.406,26.684,-44.875,-179.486,5.658,148.845
C08686=1201.401,26.933,-44.890,-179.483,5.658,148.844
C08687=1201.396,27.182,-44.906,-179.481,5.659,148.843
C08688=1201.391,27.431,-44.921,-179.478,5.659,148.843
C08689=1201.387,27.682,-44.935,-179.476,5.660,148.842
C08690=1201.382,27.931,-44.951,-179.473,5.661,148.841
C08691=1201.377,28.180,-44.966,-179.470,5.661,148.841
C08692=1201.372,28.430,-44.982,-179.468,5.662,148.840
C08693=1201.366,28.699,-44.998,-179.465,5.662,148.839
C08694=1201.361,28.967,-45.014,-179.463,5.663,148.839
C08695=1201.355,29.236,-45.031,-179.459,5.664,148.838
C08696=1201.350,29.505,-45.046,-179.457,5.665,148.837
C08697=1201.345,29.754,-45.062,-179.454,5.665,148.837
C08698=1201.340,30.003,-45.077,-179.452,5.666,148.836
C08699=1201.335,30.253,-45.093,-179.449,5.666,148.836
C08700=1201.330,30.503,-45.108,-179.447,5.667,148.835
C08701=1201.325,30.752,-45.123,-179.444,5.668,148.834
C08702=1201.320,31.001,-45.139,-179.442,5.668,148.834
C08703=1201.315,31.251,-45.153,-179.439,5.669,148.833
C08704=1201.310,31.501,-45.169,-179.437,5.669,148.832
C08705=1201.305,31.750,-45.184,-179.434,5.670,148.832
C08706=1201.300,32.000,-45.200,-179.431,5.670,148.831
C08707=1201.294,32.249,-45.215,-179.429,5.671,148.831
C08708=1201.290,32.498,-45.230,-179.426,5.672,148.830
C08709=1201.285,32.748,-45.246,-179.424,5.672,148.829
C08710=1201.280,32.997,-45.261,-179.421,5.673,148.829
C08711=1201.275,33.247,-45.277,-179.419,5.674,148.828
C08712=1201.270,33.496,-45.293,-179.416,5.674,148.827
C08713=1201.265,33.745,-45.308,-179.414,5.675,148.827
C08714=1201.260,33.995,-45.324,-179.411,5.675,148.826
C08715=1201.255,34.245,-45.339,-179.409,5.676,148.826
C08716=1201.250,34.494,-45.353,-179.406,5.677,148.825
C08717=1201.244,34.744,-45.369,-179.404,5.677,148.824
C08718=1201.240,34.994,-45.385,-179.401,5.678,148.824
C08719=1201.235,35.243,-45.400,-179.398,5.678,148.823
C08720=1201.230,35.492,-45.416,-179.396,5.679,148.822
C08721=1201.225,35.741,-45.432,-179.394,5.680,148.822
C08722=1201.221,35.991,-45.447,-179.391,5.680,148.821
C08723=1201.215,36.240,-45.463,-179.388,5.681,148.820
C08724=1201.210,36.490,-45.478,-179.386,5.682,148.820
C08725=1201.205,36.739,-45.493,-179.383,5.682,148.819
C08726=1201.200,36.989,-45.509,-179.381,5.683,148.819
C08727=1201.195,37.238,-45.525,-179.378,5.684,148.818
C08728=1201.190,37.488,-45.540,-179.375,5.685,148.818
C08729=1201.185,37.738,-45.556,-179.373,5.686,148.817
C08730=1201.180,37.987,-45.571,-179.370,5.686,148.816
C08731=1201.175,38.236,-45.587,-179.368,5.687,148.816
C08732=1201.169,38.486,-45.603,-179.365,5.687,148.815
C08733=1201.165,38.736,-45.618,-179.363,5.688,148.814
C08734=1201.160,38.984,-45.634,-179.360,5.689,148.814
C08735=1201.155,39.234,-45.650,-179.357,5.689,148.813
C08736=1201.150,39.484,-45.666,-179.355,5.690,148.813
C08737=1201.145,39.733,-45.681,-179.353,5.690,148.812
C08738=1201.140,39.982,-45.696,-179.350,5.691,148.811
C08739=1201.135,40.233,-45.712,-179.347,5.692,148.811
C08740=1201.130,40.481,-45.729,-179.345,5.692,148.810
C08741=1201.125,40.731,-45.744,-179.343,5.693,148.809
C08742=1201.121,40.981,-45.760,-179.340,5.693,148.809
C08743=1201.115,41.230,-45.775,-179.337,5.694,148.808
C08744=1201.110,41.479,-45.791,-179.335,5.695,148.808
C08745=1201.105,41.729,-45.807,-179.332,5.696,148.807
C08746=1201.100,41.978,-45.823,-179.329,5.697,148.806
C08747=1201.095,42.228,-45.839,-179.327,5.697,148.806
C08748=1201.091,42.477,-45.854,-179.324,5.698,148.805
C08749=1201.086,42.726,-45.870,-179.322,5.699,148.805
C08750=1201.080,42.976,-45.886,-179.319,5.699,148.804
C08751=1201.075,43.226,-45.902,-179.317,5.700,148.803
C08752=1201.070,43.475,-45.917,-179.314,5.701,148.803
C08753=1201.065,43.725,-45.934,-179.312,5.701,148.802
C08754=1201.060,43.974,-45.950,-179.309,5.702,148.801
C08755=1201.055,44.223,-45.965,-179.306,5.702,148.801
C08756=1201.051,44.473,-45.981,-179.304,5.703,148.800
C08757=1201.046,44.722,-45.997,-179.302,5.704,148.800
C08758=1201.041,44.972,-46.013,-179.298,5.705,148.799
C08759=1201.036,45.221,-46.029,-179.296,5.706,148.798
C08760=1201.030,45.470,-46.045,-179.294,5.706,148.798
C08761=1201.026,45.720,-46.061,-179.291,5.707,148.797
C08762=1201.020,45.969,-46.077,-179.288,5.708,148.797
C08763=1201.016,46.219,-46.093,-179.286,5.708,148.796
C08764=1201.011,46.468,-46.109,-179.284,5.709,148.795
C08765=1201.005,46.717,-46.125,-179.281,5.709,148.795
C08766=1201.000,46.968,-46.141,-179.278,5.710,148.794
C08767=1200.995,47.216,-46.157,-179.276,5.711,148.794
C08768=1200.991,47.466,-46.172,-179.274,5.711,148.793
C08769=1200.986,47.715,-46.189,-179.270,5.713,148.792
C08770=1200.981,47.965,-46.205,-179.268,5.713,148.792
C08771=1200.976,48.214,-46.221,-179.266,5.714,148.791
C08772=1200.972,48.464,-46.237,-179.263,5.715,148.791
C08773=1200.966,48.713,-46.253,-179.260,5.715,148.790
C08774=1200.961,48.962,-46.269,-179.258,5.716,148.789
C08775=1200.956,49.212,-46.285,-179.255,5.717,148.789
C08776=1200.951,49.461,-46.301,-179.253,5.717,148.788
C08777=1200.946,49.711,-46.317,-179.250,5.718,148.787
C08778=1200.941,49.960,-46.333,-179.247,5.720,148.787
C08779=1200.937,50.210,-46.349,-179.245,5.720,148.786
C08780=1200.931,50.459,-46.366,-179.242,5.721,148.786
C08781=1200.926,50.709,-46.383,-179.240,5.721,148.785
C08782=1200.921,50.958,-46.399,-179.237,5.722,148.785
C08783=1200.916,51.207,-46.415,-179.235,5.723,148.784
C08784=1200.911,51.457,-46.431,-179.232,5.723,148.783
C08785=1200.907,51.706,-46.447,-179.230,5.724,148.783
C08786=1200.901,51.956,-46.463,-179.227,5.725,148.782
C08787=1200.897,52.205,-46.480,-179.224,5.726,148.781
C08788=1200.892,52.454,-46.496,-179.222,5.726,148.781
C08789=1200.887,52.704,-46.512,-179.219,5.727,148.780
C08790=1200.882,52.954,-46.529,-179.217,5.728,148.780
C08791=1200.877,53.203,-46.544,-179.214,5.728,148.779
C08792=1200.872,53.452,-46.561,-179.212,5.729,148.779
C08793=1200.867,53.701,-46.577,-179.209,5.730,148.778
C08794=1200.862,53.952,-46.594,-179.207,5.730,148.777
C08795=1200.857,54.200,-46.610,-179.203,5.732,148.777
C08796=1200.852,54.450,-46.627,-179.201,5.733,148.776
C08797=1200.847,54.718,-46.644,-179.199,5.733,148.775
C08798=1200.841,54.986,-46.661,-179.196,5.734,148.775
C08799=1200.837,55.255,-46.679,-179.193,5.735,148.774
C08800=1200.831,55.524,-46.697,-179.190,5.736,148.773
C08801=1200.826,55.774,-46.713,-179.188,5.736,148.773
C08802=1200.821,56.022,-46.729,-179.185,5.737,148.772
C08803=1200.816,56.272,-46.746,-179.183,5.738,148.772
C08804=1200.812,56.521,-46.763,-179.180,5.739,148.771
C08805=1200.806,56.771,-46.779,-179.177,5.740,148.771
C08806=1200.801,57.021,-46.796,-179.175,5.740,148.770
C08807=1200.796,57.269,-46.812,-179.172,5.741,148.769
C08808=1200.792,57.519,-46.829,-179.170,5.741,148.769
C08809=1200.787,57.769,-46.845,-179.167,5.742,148.768
C08810=1200.781,58.018,-46.861,-179.165,5.743,148.767
C08811=1200.776,58.268,-46.878,-179.162,5.744,148.767
C08812=1200.771,58.516,-46.894,-179.159,5.745,148.766
C08813=1200.767,58.766,-46.911,-179.157,5.746,148.766
C08814=1200.762,59.016,-46.928,-179.154,5.746,148.765
C08815=1200.756,59.265,-46.944,-179.152,5.747,148.765
C08816=1200.752,59.515,-46.961,-179.149,5.748,148.764
C08817=1200.747,59.763,-46.977,-179.146,5.749,148.763
C08818=1200.742,60.013,-46.994,-179.144,5.750,148.763
C08819=1200.737,60.263,-47.011,-179.141,5.751,148.762
C08820=1200.732,60.511,-47.027,-179.139,5.751,148.761
C08821=1200.727,60.761,-47.044,-179.137,5.752,148.761
C08822=1200.722,61.011,-47.061,-179.134,5.752,148.760
C08823=1200.717,61.260,-47.077,-179.131,5.754,148.760
C08824=1200.712,61.510,-47.093,-179.128,5.754,148.759
C08825=1200.707,61.759,-47.111,-179.126,5.755,148.759
C08826=1200.702,62.008,-47.127,-179.123,5.756,148.758
C08827=1200.698,62.258,-47.144,-179.121,5.756,148.757
C08828=1200.692,62.507,-47.161,-179.119,5.757,148.757
C08829=1200.687,62.756,-47.177,-179.115,5.759,148.756
C08830=1200.683,63.006,-47.194,-179.113,5.759,148.756
C08831=1200.678,63.255,-47.211,-179.111,5.760,148.755
C08832=1200.673,63.505,-47.228,-179.108,5.761,148.754
C08833=1200.667,63.754,-47.245,-179.105,5.761,148.754
C08834=1200.663,64.004,-47.261,-179.103,5.763,148.753
C08835=1200.658,64.253,-47.278,-179.100,5.763,148.753
C08836=1200.653,64.502,-47.295,-179.097,5.764,148.752
C08837=1200.648,64.752,-47.312,-179.095,5.765,148.752
C08838=1200.644,65.001,-47.328,-179.093,5.765,148.751
C08839=1200.638,65.251,-47.345,-179.090,5.766,148.750
C08840=1200.633,65.500,-47.362,-179.087,5.768,148.750
C08841=1200.628,65.749,-47.379,-179.085,5.768,148.749
C08842=1200.624,65.999,-47.396,-179.082,5.769,148.749
C08843=1200.619,66.248,-47.413,-179.080,5.770,148.748
C08844=1200.614,66.497,-47.430,-179.077,5.770,148.747
C08845=1200.609,66.746,-47.447,-179.074,5.772,148.747
C08846=1200.604,66.996,-47.464,-179.072,5.773,148.746
C08847=1200.599,67.246,-47.481,-179.069,5.773,148.746
C08848=1200.594,67.495,-47.497,-179.067,5.774,148.745
C08849=1200.589,67.744,-47.514,-179.064,5.775,148.745
C08850=1200.584,67.994,-47.531,-179.061,5.776,148.744
C08851=1200.580,68.243,-47.549,-179.059,5.777,148.743
C08852=1200.574,68.492,-47.566,-179.056,5.777,148.743
C08853=1200.569,68.741,-47.582,-179.054,5.778,148.742
C08854=1200.564,68.991,-47.600,-179.051,5.780,148.742
C08855=1200.560,69.241,-47.616,-179.048,5.780,148.741
C08856=1200.555,69.490,-47.634,-179.046,5.781,148.740
C08857=1200.550,69.739,-47.651,-179.044,5.782,148.740
C08858=1200.545,69.989,-47.668,-179.041,5.782,148.739
C08859=1200.540,70.238,-47.685,-179.038,5.784,148.739
C08860=1200.535,70.487,-47.703,-179.036,5.785,148.738
C08861=1200.531,70.737,-47.719,-179.033,5.785,148.738
C08862=1200.525,70.986,-47.736,-179.030,5.786,148.737
C08863=1200.520,71.235,-47.753,-179.028,5.787,148.736
C08864=1200.515,71.484,-47.771,-179.025,5.788,148.736
C08865=1200.511,71.734,-47.787,-179.022,5.788,148.735
C08866=1200.506,71.984,-47.805,-179.020,5.789,148.735
C08867=1200.501,72.233,-47.822,-179.018,5.790,148.734
C08868=1200.496,72.482,-47.839,-179.014,5.791,148.733
C08869=1200.491,72.731,-47.856,-179.012,5.792,148.733
C08870=1200.486,72.981,-47.873,-179.010,5.793,148.732
C08871=1200.481,73.230,-47.891,-179.008,5.794,148.732
C08872=1200.476,73.480,-47.908,-179.004,5.795,148.731
C08873=1200.472,73.729,-47.926,-179.002,5.796,148.731
C08874=1200.467,73.979,-47.943,-179.000,5.797,148.730
C08875=1200.461,74.227,-47.959,-178.997,5.797,148.729
C08876=1200.457,74.477,-47.977,-178.994,5.798,148.729
C08877=1200.451,74.726,-47.994,-178.992,5.799,148.728
C08878=1200.447,74.976,-48.011,-178.989,5.800,148.728
C08879=1200.442,75.225,-48.029,-178.987,5.801,148.727
C08880=1200.437,75.475,-48.046,-178.984,5.802,148.727
C08881=1200.433,75.724,-48.064,-178.981,5.803,148.726
C08882=1200.427,75.973,-48.081,-178.979,5.804,148.726
C08883=1200.422,76.223,-48.099,-178.976,5.804,148.725
C08884=1200.417,76.471,-48.115,-178.973,5.806,148.724
C08885=1200.412,76.721,-48.133,-178.971,5.807,148.724
C08886=1200.407,76.970,-48.150,-178.968,5.807,148.723
C08887=1200.403,77.219,-48.168,-178.966,5.808,148.723
C08888=1200.398,77.469,-48.185,-178.963,5.809,148.722
C08889=1200.393,77.718,-48.203,-178.960,5.810,148.721
C08890=1200.388,77.968,-48.220,-178.958,5.811,148.721
C08891=1200.383,78.217,-48.238,-178.956,5.811,148.720
C08892=1200.378,78.467,-48.255,-178.953,5.813,148.720
C08893=1200.373,78.716,-48.273,-178.950,5.814,148.719
C08894=1200.368,78.966,-48.290,-178.948,5.814,148.719
C08895=1200.364,79.214,-48.308,-178.945,5.816,148.718
C08896=1200.359,79.464,-48.325,-178.942,5.817,148.718
C08897=1200.354,79.713,-48.343,-178.940,5.817,148.717
C08898=1200.349,79.963,-48.361,-178.937,5.818,148.716
C08899=1200.344,80.212,-48.377,-178.934,5.819,148.716
C08900=1200.340,80.461,-48.395,-178.932,5.820,148.715
C08901=1200.334,80.729,-48.414,-178.929,5.821,148.715
C08902=1200.328,80.998,-48.433,-178.926,5.822,148.714
C08903=1200.323,81.267,-48.452,-178.924,5.823,148.713
C08904=1200.318,81.535,-48.471,-178.920,5.824,148.713
C08905=1200.313,81.785,-48.489,-178.918,5.825,148.712
C08906=1200.309,82.033,-48.506,-178.916,5.826,148.712
C08907=1200.304,82.283,-48.524,-178.913,5.827,148.711
C08908=1200.299,82.532,-48.542,-178.910,5.828,148.711
C08909=1200.294,82.782,-48.559,-178.908,5.829,148.710
C08910=1200.289,83.031,-48.577,-178.905,5.830,148.710
C08911=1200.284,83.280,-48.595,-178.902,5.831,148.709
C08912=1200.279,83.529,-48.612,-178.900,5.832,148.708
C08913=1200.274,83.779,-48.630,-178.898,5.832,148.708
C08914=1200.269,84.028,-48.648,-178.895,5.834,148.707
C08915=1200.265,84.277,-48.666,-178.892,5.835,148.707
C08916=1200.259,84.527,-48.683,-178.890,5.835,148.706
C08917=1200.254,84.776,-48.701,-178.887,5.837,148.706
C08918=1200.249,85.025,-48.719,-178.884,5.838,148.705
C08919=1200.245,85.274,-48.737,-178.882,5.838,148.705
C08920=1200.239,85.524,-48.754,-178.879,5.840,148.704
C08921=1200.234,85.773,-48.772,-178.876,5.840,148.703
C08922=1200.230,86.022,-48.790,-178.874,5.841,148.703
C08923=1200.226,86.272,-48.808,-178.872,5.842,148.702
C08924=1200.221,86.521,-48.826,-178.869,5.844,148.702
C08925=1200.216,86.770,-48.844,-178.866,5.844,148.701
C08926=1200.211,87.020,-48.861,-178.864,5.845,148.701
C08927=1200.206,87.269,-48.879,-178.861,5.846,148.700
C08928=1200.201,87.519,-48.897,-178.858,5.847,148.699
C08929=1200.196,87.768,-48.915,-178.856,5.848,148.699
C08930=1200.191,88.017,-48.933,-178.853,5.849,148.698
C08931=1200.186,88.266,-48.951,-178.851,5.850,148.698
C08932=1200.181,88.515,-48.969,-178.848,5.851,148.697
C08933=1200.177,88.764,-48.987,-178.846,5.853,148.697
C08934=1200.172,89.014,-49.005,-178.843,5.853,148.696
C08935=1200.167,89.264,-49.023,-178.840,5.854,148.696
C08936=1200.162,89.513,-49.041,-178.838,5.855,148.695
C08937=1200.157,89.762,-49.059,-178.835,5.856,148.695
C08938=1200.152,90.012,-49.077,-178.833,5.857,148.694
C08939=1200.147,90.261,-49.095,-178.830,5.858,148.693
C08940=1200.142,90.510,-49.112,-178.828,5.859,148.693
C08941=1200.138,90.759,-49.130,-178.825,5.860,148.692
C08942=1200.133,91.009,-49.149,-178.822,5.862,148.692
C08943=1200.128,91.258,-49.167,-178.820,5.862,148.691
C08944=1200.123,91.508,-49.185,-178.817,5.863,148.691
C08945=1200.118,91.757,-49.203,-178.814,5.864,148.690
C08946=1200.113,92.006,-49.221,-178.812,5.865,148.690
C08947=1200.108,92.255,-49.239,-178.809,5.866,148.689
C08948=1200.104,92.505,-49.258,-178.806,5.867,148.689
C08949=1200.099,92.754,-49.276,-178.804,5.868,148.688
C08950=1200.094,93.003,-49.294,-178.801,5.870,148.687
C08951=1200.089,93.252,-49.312,-178.799,5.871,148.687
C08952=1200.084,93.501,-49.330,-178.796,5.871,148.686
C08953=1200.080,93.751,-49.349,-178.793,5.873,148.686
C08954=1200.074,94.001,-49.367,-178.791,5.873,148.685
C08955=1200.069,94.250,-49.385,-178.788,5.874,148.685
C08956=1200.064,94.499,-49.403,-178.786,5.876,148.684
C08957=1200.060,94.748,-49.421,-178.783,5.876,148.684
C08958=1200.056,94.997,-49.440,-178.781,5.877,148.683
C08959=1200.051,95.246,-49.458,-178.778,5.879,148.683
C08960=1200.045,95.496,-49.477,-178.775,5.880,148.682
C08961=1200.040,95.745,-49.495,-178.772,5.881,148.682
C08962=1200.036,95.995,-49.513,-178.770,5.882,148.681
C08963=1200.031,96.244,-49.531,-178.768,5.882,148.680
C08964=1200.026,96.493,-49.550,-178.765,5.884,148.680
C08965=1200.021,96.742,-49.568,-178.762,5.885,148.679
C08966=1200.016,96.992,-49.587,-178.760,5.886,148.679
C08967=1200.011,97.241,-49.605,-178.757,5.887,148.678
C08968=1200.007,97.490,-49.623,-178.755,5.888,148.678
C08969=1200.002,97.739,-49.641,-178.752,5.889,148.677
C08970=1199.997,97.989,-49.660,-178.749,5.890,148.677
C08971=1199.992,98.238,-49.678,-178.747,5.891,148.676
C08972=1199.987,98.487,-49.697,-178.744,5.892,148.676
C08973=1199.982,98.736,-49.715,-178.741,5.893,148.675
C08974=1199.977,98.986,-49.734,-178.739,5.894,148.674
C08975=1199.973,99.235,-49.753,-178.736,5.896,148.674
C08976=1199.968,99.484,-49.771,-178.734,5.896,148.673
C08977=1199.964,99.734,-49.789,-178.731,5.898,148.673
C08978=1199.958,99.983,-49.808,-178.728,5.899,148.672
C08979=1199.953,100.232,-49.826,-178.726,5.899,148.672
C08980=1199.948,100.481,-49.844,-178.723,5.901,148.671
C08981=1199.944,100.731,-49.864,-178.721,5.902,148.671
C08982=1199.939,100.980,-49.882,-178.718,5.903,148.670
C08983=1199.934,101.229,-49.900,-178.715,5.904,148.670
C08984=1199.929,101.479,-49.919,-178.713,5.905,148.669
C08985=1199.924,101.728,-49.937,-178.710,5.906,148.669
C08986=1199.920,101.976,-49.956,-178.708,5.907,148.668
C08987=1199.914,102.227,-49.975,-178.705,5.909,148.668
C08988=1199.910,102.476,-49.993,-178.702,5.909,148.667
C08989=1199.905,102.724,-50.012,-178.700,5.910,148.667
C08990=1199.900,102.974,-50.031,-178.697,5.912,148.666
C08991=1199.895,103.223,-50.049,-178.695,5.913,148.666
C08992=1199.890,103.473,-50.068,-178.692,5.914,148.665
C08993=1199.886,103.722,-50.087,-178.689,5.915,148.665
C08994=1199.881,103.971,-50.105,-178.686,5.916,148.664
C08995=1199.876,104.221,-50.125,-178.684,5.917,148.664
C08996=1199.871,104.470,-50.143,-178.681,5.918,148.663
C08997=1199.866,104.719,-50.162,-178.679,5.920,148.662
C08998=1199.861,104.968,-50.180,-178.676,5.920,148.662
C08999=1199.857,105.217,-50.199,-178.673,5.922,148.661
C09000=1199.852,105.467,-50.218,-178.671,5.922,148.661
C09001=1199.847,105.716,-50.237,-178.668,5.924,148.660
C09002=1199.842,105.965,-50.256,-178.666,5.925,148.660
C09003=1199.837,106.214,-50.274,-178.663,5.926,148.659
C09004=1199.832,106.463,-50.294,-178.661,5.928,148.659
C09005=1199.828,106.732,-50.313,-178.658,5.928,148.658
C09006=1199.822,107.000,-50.334,-178.655,5.929,148.658
C09007=1199.816,107.269,-50.354,-178.652,5.931,148.657
C09008=1199.812,107.537,-50.374,-178.650,5.932,148.657
C09009=1199.807,107.787,-50.393,-178.646,5.933,148.656
C09010=1199.802,108.036,-50.412,-178.644,5.934,148.656
C09011=1199.797,108.285,-50.431,-178.641,5.936,148.655
C09012=1199.792,108.534,-50.449,-178.639,5.937,148.655
C09013=1199.788,108.783,-50.469,-178.636,5.938,148.654
C09014=1199.783,109.032,-50.488,-178.634,5.939,148.653
C09015=1199.778,109.282,-50.507,-178.632,5.940,148.653
C09016=1199.773,109.531,-50.526,-178.628,5.941,148.652
C09017=1199.768,109.780,-50.545,-178.626,5.942,148.652
C09018=1199.763,110.029,-50.564,-178.623,5.944,148.651
C09019=1199.759,110.279,-50.583,-178.621,5.944,148.651
C09020=1199.753,110.528,-50.602,-178.618,5.946,148.650
C09021=1199.749,110.777,-50.621,-178.616,5.947,148.650
C09022=1199.744,111.026,-50.640,-178.612,5.948,148.649
C09023=1199.739,111.276,-50.659,-178.610,5.949,148.649
C09024=1199.734,111.525,-50.678,-178.607,5.951,148.648
C09025=1199.730,111.774,-50.698,-178.605,5.951,148.648
C09026=1199.725,112.023,-50.716,-178.602,5.953,148.647
C09027=1199.720,112.273,-50.736,-178.600,5.954,148.647
C09028=1199.715,112.522,-50.755,-178.597,5.956,148.646
C09029=1199.711,112.771,-50.774,-178.594,5.956,148.646
C09030=1199.705,113.020,-50.793,-178.592,5.957,148.645
C09031=1199.701,113.269,-50.812,-178.589,5.959,148.645
C09032=1199.696,113.518,-50.831,-178.587,5.959,148.644
C09033=1199.691,113.768,-50.851,-178.584,5.961,148.644
C09034=1199.686,114.017,-50.869,-178.582,5.962,148.643
C09035=1199.682,114.267,-50.889,-178.579,5.964,148.643
C09036=1199.676,114.515,-50.908,-178.576,5.964,148.642
C09037=1199.672,114.765,-50.927,-178.574,5.966,148.642
C09038=1199.668,115.014,-50.947,-178.571,5.967,148.641
C09039=1199.662,115.263,-50.966,-178.568,5.968,148.641
C09040=1199.657,115.513,-50.985,-178.566,5.969,148.640
C09041=1199.653,115.761,-51.004,-178.563,5.971,148.640
C09042=1199.648,116.011,-51.024,-178.561,5.972,148.639
C09043=1199.643,116.260,-51.043,-178.558,5.973,148.639
C09044=1199.638,116.509,-51.063,-178.556,5.974,148.638
C09045=1199.634,116.759,-51.082,-178.552,5.975,148.638
C09046=1199.629,117.007,-51.101,-178.550,5.976,148.637
C09047=1199.624,117.257,-51.121,-178.547,5.978,148.637
C09048=1199.619,117.506,-51.140,-178.545,5.979,148.636
C09049=1199.615,117.755,-51.159,-178.542,5.980,148.636
C09050=1199.609,118.004,-51.178,-178.540,5.981,148.635
C09051=1199.605,118.254,-51.198,-178.537,5.983,148.635
C09052=1199.600,118.503,-51.218,-178.534,5.983,148.634
C09053=1199.595,118.752,-51.236,-178.532,5.985,148.634
C09054=1199.590,119.001,-51.256,-178.530,5.986,148.633
C09055=1199.586,119.251,-51.276,-178.526,5.987,148.633
C09056=1199.580,119.500,-51.295,-178.524,5.988,148.632
C09057=1199.576,119.749,-51.315,-178.521,5.990,148.632
C09058=1199.571,119.998,-51.335,-178.519,5.991,148.631
C09059=1199.567,120.247,-51.354,-178.516,5.992,148.631
C09060=1199.562,120.496,-51.373,-178.514,5.993,148.630
C09061=1199.556,120.745,-51.393,-178.511,5.995,148.630
C09062=1199.552,120.995,-51.412,-178.508,5.995,148.629
C09063=1199.547,121.244,-51.432,-178.506,5.997,148.629
C09064=1199.542,121.493,-51.451,-178.503,5.999,148.628
C09065=1199.538,121.742,-51.471,-178.500,6.000,148.628
C09066=1199.533,121.991,-51.491,-178.498,6.001,148.627
C09067=1199.528,122.240,-51.510,-178.495,6.002,148.627
C09068=1199.523,122.490,-51.530,-178.492,6.004,148.626
C09069=1199.518,122.739,-51.549,-178.490,6.005,148.626
C09070=1199.514,122.988,-51.570,-178.487,6.006,148.625
C09071=1199.509,123.237,-51.589,-178.485,6.007,148.625
C09072=1199.504,123.487,-51.609,-178.482,6.008,148.624
C09073=1199.499,123.736,-51.628,-178.480,6.009,148.624
C09074=1199.494,123.985,-51.648,-178.477,6.011,148.623
C09075=1199.489,124.234,-51.668,-178.474,6.012,148.623
C09076=1199.485,124.483,-51.687,-178.472,6.013,148.622
C09077=1199.481,124.732,-51.707,-178.469,6.015,148.622
C09078=1199.476,124.981,-51.727,-178.466,6.016,148.621
C09079=1199.471,125.231,-51.746,-178.464,6.018,148.621
C09080=1199.466,125.480,-51.767,-178.461,6.018,148.620
C09081=1199.462,125.729,-51.786,-178.458,6.020,148.620
C09082=1199.456,125.978,-51.806,-178.456,6.021,148.620
C09083=1199.452,126.227,-51.826,-178.453,6.022,148.619
C09084=1199.447,126.477,-51.846,-178.451,6.023,148.619
C09085=1199.442,126.726,-51.865,-178.448,6.025,148.618
C09086=1199.437,126.974,-51.885,-178.445,6.026,148.618
C09087=1199.433,127.224,-51.905,-178.443,6.027,148.617
C09088=1199.428,127.473,-51.925,-178.440,6.029,148.617
C09089=1199.423,127.723,-51.945,-178.438,6.030,148.616
C09090=1199.418,127.971,-51.964,-178.435,6.032,148.616
C09091=1199.414,128.220,-51.985,-178.432,6.032,148.615
C09092=1199.409,128.470,-52.004,-178.430,6.034,148.615
C09093=1199.404,128.719,-52.025,-178.427,6.036,148.614
C09094=1199.399,128.969,-52.045,-178.424,6.036,148.614
C09095=1199.394,129.217,-52.065,-178.422,6.038,148.613
C09096=1199.389,129.467,-52.085,-178.420,6.039,148.613
C09097=1199.385,129.716,-52.105,-178.416,6.040,148.612
C09098=1199.380,129.965,-52.125,-178.414,6.041,148.612
C09099=1199.376,130.214,-52.145,-178.412,6.043,148.611
C09100=1199.370,130.463,-52.164,-178.408,6.045,148.611
C09101=1199.366,130.712,-52.185,-178.406,6.045,148.610
C09102=1199.361,130.961,-52.204,-178.404,6.047,148.610
C09103=1199.356,131.211,-52.225,-178.401,6.048,148.609
C09104=1199.351,131.460,-52.246,-178.398,6.050,148.609
C09105=1199.347,131.709,-52.265,-178.395,6.051,148.608
C09106=1199.342,131.957,-52.285,-178.393,6.052,148.608
C09107=1199.337,132.207,-52.305,-178.390,6.054,148.608
C09108=1199.332,132.456,-52.325,-178.388,6.054,148.607
C09109=1199.327,132.725,-52.347,-178.385,6.056,148.607
C09110=1199.322,132.993,-52.369,-178.382,6.058,148.606
C09111=1199.317,133.262,-52.391,-178.379,6.059,148.606
C09112=1199.312,133.531,-52.413,-178.376,6.061,148.605
C09113=1199.306,133.780,-52.433,-178.374,6.062,148.605
C09114=1199.302,134.029,-52.453,-178.371,6.063,148.604
C09115=1199.298,134.278,-52.473,-178.369,6.064,148.604
C09116=1199.293,134.527,-52.493,-178.366,6.066,148.603
C09117=1199.288,134.777,-52.514,-178.363,6.068,148.603
C09118=1199.283,135.026,-52.534,-178.361,6.069,148.602
C09119=1199.278,135.275,-52.554,-178.358,6.070,148.602
C09120=1199.274,135.524,-52.574,-178.356,6.071,148.601
C09121=1199.269,135.773,-52.595,-178.353,6.073,148.601
C09122=1199.264,136.022,-52.616,-178.350,6.074,148.600
C09123=1199.259,136.271,-52.635,-178.348,6.075,148.600
C09124=1199.255,136.520,-52.655,-178.345,6.077,148.600
C09125=1199.249,136.769,-52.676,-178.342,6.078,148.599
C09126=1199.245,137.018,-52.697,-178.340,6.079,148.599
C09127=1199.241,137.267,-52.717,-178.337,6.081,148.598
C09128=1199.235,137.517,-52.737,-178.335,6.082,148.598
C09129=1199.231,137.766,-52.758,-178.332,6.083,148.597
C09130=1199.226,138.015,-52.778,-178.329,6.085,148.597
C09131=1199.221,138.264,-52.799,-178.327,6.086,148.596
C09132=1199.217,138.513,-52.819,-178.324,6.088,148.596
C09133=1199.212,138.762,-52.840,-178.321,6.089,148.595
C09134=1199.207,139.011,-52.861,-178.319,6.090,148.595
C09135=1199.202,139.261,-52.880,-178.316,6.092,148.594
C09136=1199.198,139.510,-52.901,-178.313,6.094,148.594
C09137=1199.193,139.759,-52.922,-178.311,6.094,148.594
C09138=1199.188,140.008,-52.942,-178.308,6.096,148.593
C09139=1199.184,140.257,-52.963,-178.306,6.097,148.593
C09140=1199.179,140.506,-52.984,-178.303,6.099,148.592
C09141=1199.174,140.755,-53.004,-178.300,6.100,148.592
C09142=1199.169,141.005,-53.025,-178.298,6.101,148.591
